// TIA Portal V20 export
FUNCTION_BLOCK "CallEquipment"   // FB36, LAD
TITLE = CallEquipment
AUTHOR : ERsystem_FA2_DH. Kim
// This block contains the logic and futher calls (e.g. sequences, control modules, diagnostics etc.) of the equipment module.
// stored: IsIECCheckEnabled true, MemoryReserve 100, Namespace Unit1.Em3, SetENOAutomatically false
   VAR_INPUT
      ZoneOperationEnable { ExternalWritable := 'False'} : "LWONIK_typeSafetyZoneManualOperation";
   END_VAR
   VAR_IN_OUT
      unitStatus : "LAF_typeUnitStatus";   // Current unit status o be used in this EM
      unitAlarmDB : "LAF_typeAlarms";   // Summarized EM Alarms for the Unit
      emFeedback : "LUC_typeEmFeedback";   // Feedback of the EM to the Unit
   END_VAR
   VAR
      InstSequenceWebGuide : "Unit1.Em3.Sequence_1_WebGuide";
      instWebGuideHomeJob1 { S7_SetPoint := 'True'} : "LAF_SelectJob";
      instWebGuideGuidingJob2 { S7_SetPoint := 'True'} : "LAF_SelectJob";
      instCmSafetyPinIdlePositionSensor : "LBC_DigitalSignalCn";
      instCmIonizerTopMaintDetection { S7_SetPoint := 'True'} : "LBC_DigitalSignalCn";
      instCmIonizerTopErrorDetection { S7_SetPoint := 'True'} : "LBC_DigitalSignalCn";
      instCmIonizerBtmMaintDetection { S7_SetPoint := 'True'} : "LBC_DigitalSignalCn";
      instCmIonizerBtmErrorDetection { S7_SetPoint := 'True'} : "LBC_DigitalSignalCn";
      instCmDancerEncoder { ExternalAccessible := 'False'; ExternalVisible := 'False'; ExternalWritable := 'False'; S7_SetPoint := 'True'} : "LBC_AnalogInputCn";
      instCmLoadCellControllerInterface { ExternalAccessible := 'False'; ExternalVisible := 'False'; ExternalWritable := 'False'; S7_SetPoint := 'True'} : "LBC_AnalogInputCn";
      instCmDancerElectroPneumaticRegulator { ExternalAccessible := 'False'; ExternalVisible := 'False'; ExternalWritable := 'False'; S7_SetPoint := 'True'} : "LBC_AnalogOutputCn";
      instCmCompensatorAxisX { S7_SetPoint := 'True'} : "LBC_Axis64Pos_TecPlcCn";
      instCmUnwinderVirtualAxisX { S7_SetPoint := 'True'} : "LBC_Axis64Pos_TecPlcCn";
      instInterlockCompensatorAxisX { S7_SetPoint := 'True'} : "LER_Axis64Pos_InterlockSummary";
      instInterlockUnwinderVirtualAxisX { S7_SetPoint := 'True'} : "LER_Axis64Pos_InterlockSummary";
      instCmDancerFwdBwd { ExternalAccessible := 'False'; ExternalVisible := 'False'; ExternalWritable := 'False'; S7_SetPoint := 'True'} : "LBC_TwoWayActuatorCn";
      instCmSepaUnwinderIonizerTop { ExternalAccessible := 'False'; ExternalVisible := 'False'; ExternalWritable := 'False'; S7_SetPoint := 'True'} : "LBC_TwoWayActuatorCn";
      instCmSepaUnwinderIonizerBottom { ExternalAccessible := 'False'; ExternalVisible := 'False'; ExternalWritable := 'False'; S7_SetPoint := 'True'} : "LBC_TwoWayActuatorCn";
      instCmEpcPivot { ExternalAccessible := 'False'; ExternalVisible := 'False'; ExternalWritable := 'False'; S7_SetPoint := 'True'} : "LER_EPC_CON600";
      instManageAlarms { ExternalWritable := 'False'} : "LAF_ManageAlarms";
      instEventsPFE : "Unit1.Em3.EventsPFE";
      statUnitStatus { ExternalWritable := 'False'} : "LAF_typeUnitStatus";   // Unit Status used in this EM
      statSlmStatus : Struct
         running { ExternalWritable := 'False'} : Bool;
         powerOff { ExternalWritable := 'False'} : Bool;
      END_STRUCT;
      statTonTime { ExternalAccessible := 'False'; ExternalVisible := 'False'; ExternalWritable := 'False'} : Array[0..1999] of TON_TIME;
      statTofTime { ExternalAccessible := 'False'; ExternalVisible := 'False'; ExternalWritable := 'False'} : Array[0..99] of TOF_TIME;
      statPulse { ExternalAccessible := 'False'; ExternalVisible := 'False'; ExternalWritable := 'False'} : Struct
         miscellaneous : Array[0..99] of Bool;
         workingDone : Struct
            mainPnP : Array[0..99] of Bool;
            alignTable : Array[0..99] of Bool;
            ngPnP : Array[0..99] of Bool;
         END_STRUCT;
         axisEnable : Array[0..99] of Bool;
         brakeTest : Array[0..99] of Bool;
      END_STRUCT;
      statEnableManualCmds : Bool;
      Scan_on : Bool;
      "*** Interlock Axis ***" { ExternalAccessible := 'False'; ExternalVisible := 'False'; ExternalWritable := 'False'} : Bool;
      "compenastor X Home" { S7_SetPoint := 'True'} : "Homing.LER_Axis";
      "compenastor X Jog_CW" { S7_SetPoint := 'True'} : "Jog.LER_Axis";
      "compenastor X Jog_CCW" { S7_SetPoint := 'True'} : "Jog.LER_Axis";
      "compenastor X Position_" { S7_SetPoint := 'True'} : Array[0..5] of "Position.LER_Axis";
      "*** Interlock Actuator ******" { ExternalAccessible := 'False'; ExternalVisible := 'False'; ExternalWritable := 'False'} : Bool;
      "DancerFwdBwd Home" { S7_SetPoint := 'True'} : "Cylinder.LER_Actuator";
      "DancerFwdBwd Work" { S7_SetPoint := 'True'} : "Cylinder.LER_Actuator";
      "SepaUnwinderIonizer Home" { S7_SetPoint := 'True'} : "Cylinder.LER_Actuator";
      "SepaUnwinderIonizer Work" { S7_SetPoint := 'True'} : "Cylinder.LER_Actuator";
      "SepaUnwinderIonizerBottom Home" { S7_SetPoint := 'True'} : "Cylinder.LER_Actuator";
      "SepaUnwinderIonizerBottom Work" { S7_SetPoint := 'True'} : "Cylinder.LER_Actuator";
      AXIS3 : "LER_CM_Name";
      Cylinder10 : "LER_CM_Name";
      instCmRotaionSafetyPinPositionSensor { ExternalAccessible := 'False'; ExternalVisible := 'False'; ExternalWritable := 'False'} : "LBC_DigitalSignalCn";
      citi_Ptrig : Array[0..20] of Bool;
      citiTon : Array[0..20] of TON_TIME;
      citi : Time;
      citiTest : Array[0..20] of Bool;
   END_VAR
   VAR_TEMP
      tempIndex : Int;
      tempScInProduction : Bool;   // Mode Production and StateComplete
      tempScNoProduction : Bool;   // Mode Manual and StateComplete
   END_VAR
   VAR CONSTANT
      delayTime : Time := T#3s;
      TRUE : Bool := TRUE;
      FALSE : Bool := FALSE;
      NO_JOB : DInt;   // No job
      MIN_POSITION_NUMBER : SInt;
      INIT_POSITION_NUMBER : SInt := -1;
   END_VAR
   // // instCmCompensatorAxisX.instAxisCtrl.configuration.posAbsolute.positionChangeOnTheFly : TRUE: Changing position on-the-fly; FALSE: Position change requires a new rising edge at source.posAbsolute input
   // // instCmCompensatorAxisX.instAxisCtrl.configuration.posAbsolute.velocityChangeOnTheFly : TRUE: Changing velocity on-the-fly; FALSE: Velocity change requires a new rising edge at source.posAbsolute input
   // // instCmCompensatorAxisX.statCurrentInputs.posAbsolute : Internal storage for edge detection of source.posAbsolute
   // // instCmCompensatorAxisX.statPreviousInputs.posAbsolute : Internal storage for edge detection of source.posAbsolute
   // // instCmCompensatorAxisX.statCurrentInterface.posAbsolute : Internal storage for edge detection of source.posAbsolute
   // // instCmCompensatorAxisX.statPreviousInterface.posAbsolute : Internal storage for edge detection of source.posAbsolute
   // // instCmUnwinderVirtualAxisX.instAxisCtrl.configuration.posAbsolute.positionChangeOnTheFly : TRUE: Changing position on-the-fly; FALSE: Position change requires a new rising edge at source.posAbsolute input
   // // instCmUnwinderVirtualAxisX.instAxisCtrl.configuration.posAbsolute.velocityChangeOnTheFly : TRUE: Changing velocity on-the-fly; FALSE: Velocity change requires a new rising edge at source.posAbsolute input
   // // instCmUnwinderVirtualAxisX.statCurrentInputs.posAbsolute : Internal storage for edge detection of source.posAbsolute
   // // instCmUnwinderVirtualAxisX.statPreviousInputs.posAbsolute : Internal storage for edge detection of source.posAbsolute
   // // instCmUnwinderVirtualAxisX.statCurrentInterface.posAbsolute : Internal storage for edge detection of source.posAbsolute
   // // instCmUnwinderVirtualAxisX.statPreviousInterface.posAbsolute : Internal storage for edge detection of source.posAbsolute
   VAR_TEMP   // added for the SCL form of the ladder/FBD networks
      _w1 : Bool;
      _w2 : Bool;
      _w3 : Bool;
      _w4 : Bool;
      _w5 : Bool;
      _w6 : Bool;
      _w7 : Bool;
      _w8 : Bool;
      _w9 : Bool;
   END_VAR
BEGIN

REGION Network 1: BLOCK INFO HEADER
   // (company) / (C) Copyright (year)
   // ---------------------------------------------------------------------------------
   // Title:                             (Title of this block)
   // Comment/Function: (that is implemented in the block)
   // Library/Family:           (that the source is dedicated to)
   // Author:                        (department / person in charge / contact)
   // Target System:          (test system with FW version)
   // Engineering:              TIA Portal (SW version)
   // Restrictions:               (OB types, etc.)
   // Requirements:           (hardware, technological package, etc.)
   // ---------------------------------------------------------------------------------
   // Change log table:
   // Version          | Date             | Signature      | Expert in charge  | Changes applied ------------------------|----------------------|-------------------------|--------------------------------|-----------------------
   // 001.000.000 | yyyy-mm-dd | 0x00000000 | (name of expert) | First released version
END_REGION

REGION Network 2: DESCRIPTION
   // This is a template block provided by the Automation Framework. It can be used to create an own project.
   // The Block Info Header is prepared to put in your own data.
   // Description of the block could be added here and the docu created by Code2Docu.
END_REGION

REGION Network 3: TRUE: Disable the monitoring of the Home position feedback. FALSE: Home position is reached after `monitoringReachingFeedback` time expires.
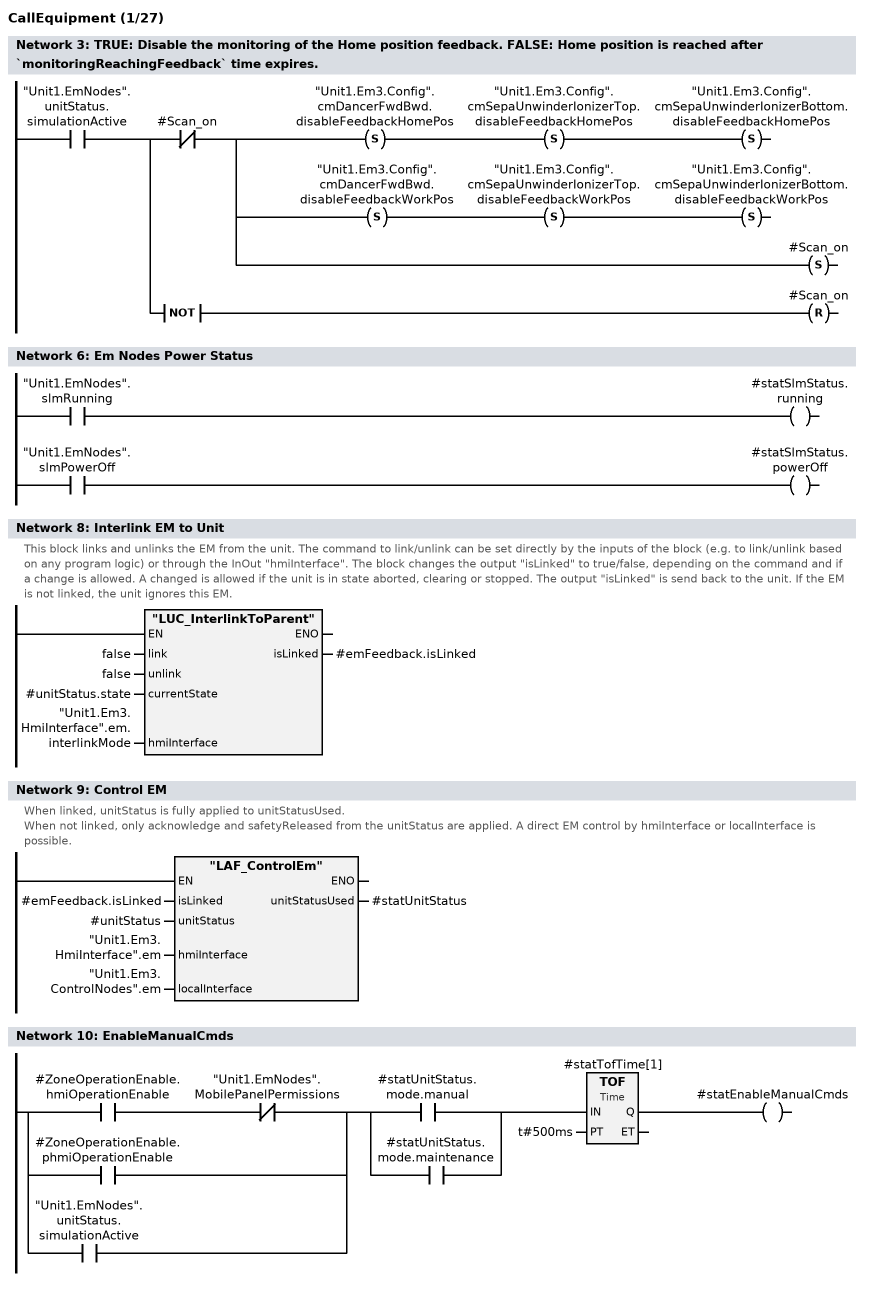
   RUNG wire#powerrail
      Contact( "Unit1.EmNodes".unitStatus.simulationActive )
      wire#w1
      I_Contact( #Scan_on )
      wire#w2
      S_Coil( "Unit1.Em3.Config".cmDancerFwdBwd.disableFeedbackHomePos )
      S_Coil( "Unit1.Em3.Config".cmSepaUnwinderIonizerTop.disableFeedbackHomePos )
      S_Coil( "Unit1.Em3.Config".cmSepaUnwinderIonizerBottom.disableFeedbackHomePos )
   END_RUNG
   RUNG wire#w2
      S_Coil( "Unit1.Em3.Config".cmDancerFwdBwd.disableFeedbackWorkPos )
      S_Coil( "Unit1.Em3.Config".cmSepaUnwinderIonizerTop.disableFeedbackWorkPos )
      S_Coil( "Unit1.Em3.Config".cmSepaUnwinderIonizerBottom.disableFeedbackWorkPos )
   END_RUNG
   RUNG wire#w2
      S_Coil( #Scan_on )
   END_RUNG
   RUNG wire#w1
      Not()
      R_Coil( #Scan_on )
   END_RUNG
   // the same network as SCL:
   IF "Unit1.EmNodes".unitStatus.simulationActive AND NOT #Scan_on THEN
       "Unit1.Em3.Config".cmDancerFwdBwd.disableFeedbackHomePos := TRUE;
       "Unit1.Em3.Config".cmSepaUnwinderIonizerTop.disableFeedbackHomePos := TRUE;
       "Unit1.Em3.Config".cmSepaUnwinderIonizerBottom.disableFeedbackHomePos := TRUE;
       "Unit1.Em3.Config".cmDancerFwdBwd.disableFeedbackWorkPos := TRUE;
       "Unit1.Em3.Config".cmSepaUnwinderIonizerTop.disableFeedbackWorkPos := TRUE;
       "Unit1.Em3.Config".cmSepaUnwinderIonizerBottom.disableFeedbackWorkPos := TRUE;
       #Scan_on := TRUE;
   END_IF;
   IF NOT "Unit1.EmNodes".unitStatus.simulationActive THEN #Scan_on := FALSE; END_IF;
END_REGION

REGION Network 4: ******************** Unit Input ********************
END_REGION

REGION Network 5: Em2 Sequence Interface
END_REGION

REGION Network 6: Em Nodes Power Status
   RUNG wire#powerrail
      Contact( "Unit1.EmNodes".slmRunning )
      Coil( #statSlmStatus.running )
   END_RUNG
   RUNG wire#powerrail
      Contact( "Unit1.EmNodes".slmPowerOff )
      Coil( #statSlmStatus.powerOff )
   END_RUNG
   // the same network as SCL:
   #statSlmStatus.running := "Unit1.EmNodes".slmRunning;
   #statSlmStatus.powerOff := "Unit1.EmNodes".slmPowerOff;
END_REGION

REGION Network 7: *************** Equipment Control **************************
END_REGION

REGION Network 8: Interlink EM to Unit
   // This block links and unlinks the EM from the unit. The command to link/unlink can be set directly by the inputs of the block (e.g. to link/unlink based on any program logic) or through the InOut "hmiInterface". The block changes the output "isLinked" to true/false, depending on the command and if a change is allowed. A changed is allowed if the unit is in state aborted, clearing or stopped. The output "isLinked" is send back to the unit. If the EM is not linked, the unit ignores this EM.
   RUNG wire#powerrail
      "LUC_InterlinkToParent"(link := false, unlink := false, currentState := #unitStatus.state, hmiInterface := "Unit1.Em3.HmiInterface".em.interlinkMode, isLinked => #emFeedback.isLinked)
   END_RUNG
   // the same network as SCL:
   "LUC_InterlinkToParent"(link := false,
                           unlink := false,
                           currentState := #unitStatus.state,
                           hmiInterface := "Unit1.Em3.HmiInterface".em.interlinkMode,
                           isLinked => #emFeedback.isLinked);
END_REGION

REGION Network 9: Control EM
   // When linked, unitStatus is fully applied to unitStatusUsed.
   // When not linked, only acknowledge and safetyReleased from the unitStatus are applied. A direct EM control by hmiInterface or localInterface is possible.
   RUNG wire#powerrail
      "LAF_ControlEm"(isLinked := #emFeedback.isLinked, unitStatus := #unitStatus, hmiInterface := "Unit1.Em3.HmiInterface".em, localInterface := "Unit1.Em3.ControlNodes".em, unitStatusUsed => #statUnitStatus)
   END_RUNG
   // the same network as SCL:
   "LAF_ControlEm"(isLinked := #emFeedback.isLinked,
                   unitStatus := #unitStatus,
                   hmiInterface := "Unit1.Em3.HmiInterface".em,
                   localInterface := "Unit1.Em3.ControlNodes".em,
                   unitStatusUsed => #statUnitStatus);
END_REGION

REGION Network 10: EnableManualCmds
   RUNG wire#powerrail
      Contact( #ZoneOperationEnable.hmiOperationEnable )
      I_Contact( "Unit1.EmNodes".MobilePanelPermissions )
      wire#w1
      Contact( #statUnitStatus.mode.manual )
      wire#w2
      { S7_Templates := "time_type := Time" } #statTofTime[1].TOF(pt := t#500ms, et =>)
      Coil( #statEnableManualCmds )
   END_RUNG
   RUNG wire#powerrail
      Contact( #ZoneOperationEnable.phmiOperationEnable )
   END_RUNG wire#w1
   RUNG wire#powerrail
      Contact( "Unit1.EmNodes".unitStatus.simulationActive )
   END_RUNG wire#w1
   RUNG wire#w1
      Contact( #statUnitStatus.mode.maintenance )
   END_RUNG wire#w2
   // the same network as SCL:
   #statTofTime[1].TOF(IN := ((#ZoneOperationEnable.hmiOperationEnable AND NOT "Unit1.EmNodes".MobilePanelPermissions) OR #ZoneOperationEnable.phmiOperationEnable OR "Unit1.EmNodes".unitStatus.simulationActive) AND (#statUnitStatus.mode.manual OR #statUnitStatus.mode.maintenance),
                       PT := t#500ms);
   #statEnableManualCmds := #statTofTime[1].Q;
END_REGION

REGION Network 11: *************** Control Modules (Sensors) ********************
   // Call control modules that are sensors before the em logic (jobs and sequence), so that the latest value is used in the logic.
END_REGION

REGION Network 12: Call cmDancer Safety Pin Idle Position Sensor (LBC_DigitalSignal)
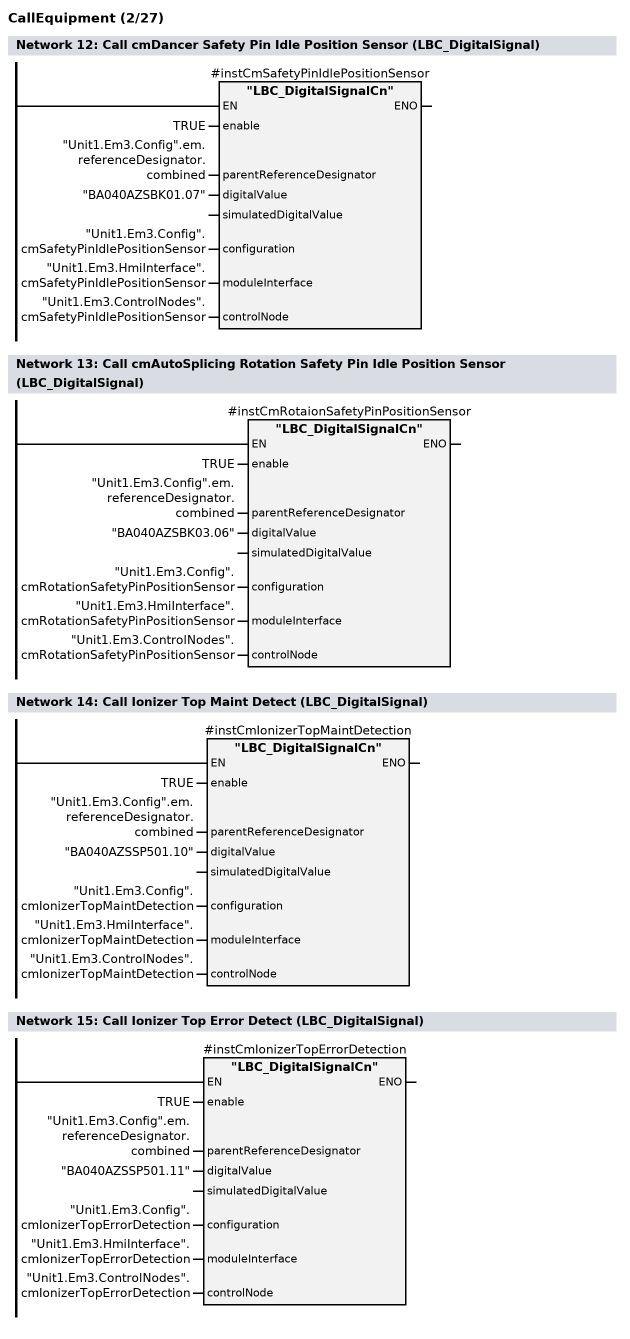
   RUNG wire#powerrail
      #instCmSafetyPinIdlePositionSensor(enable := TRUE, parentReferenceDesignator := "Unit1.Em3.Config".em.referenceDesignator.combined, digitalValue := "BA040AZSBK01.07", simulatedDigitalValue :=, configuration := "Unit1.Em3.Config".cmSafetyPinIdlePositionSensor, moduleInterface := "Unit1.Em3.HmiInterface".cmSafetyPinIdlePositionSensor, controlNode := "Unit1.Em3.ControlNodes".cmSafetyPinIdlePositionSensor)
   END_RUNG
   // the same network as SCL:
   #instCmSafetyPinIdlePositionSensor(enable := TRUE,   // "LBC_DigitalSignalCn"
                           parentReferenceDesignator := "Unit1.Em3.Config".em.referenceDesignator.combined,
                           digitalValue := "BA040AZSBK01.07",
                           configuration := "Unit1.Em3.Config".cmSafetyPinIdlePositionSensor,
                           moduleInterface := "Unit1.Em3.HmiInterface".cmSafetyPinIdlePositionSensor,
                           controlNode := "Unit1.Em3.ControlNodes".cmSafetyPinIdlePositionSensor);
END_REGION

REGION Network 13: Call cmAutoSplicing Rotation Safety Pin Idle Position Sensor (LBC_DigitalSignal)
   RUNG wire#powerrail
      #instCmRotaionSafetyPinPositionSensor(enable := TRUE, parentReferenceDesignator := "Unit1.Em3.Config".em.referenceDesignator.combined, digitalValue := "BA040AZSBK03.06", simulatedDigitalValue :=, configuration := "Unit1.Em3.Config".cmRotationSafetyPinPositionSensor, moduleInterface := "Unit1.Em3.HmiInterface".cmRotationSafetyPinPositionSensor, controlNode := "Unit1.Em3.ControlNodes".cmRotationSafetyPinPositionSensor)
   END_RUNG
   // the same network as SCL:
   #instCmRotaionSafetyPinPositionSensor(enable := TRUE,   // "LBC_DigitalSignalCn"
                           parentReferenceDesignator := "Unit1.Em3.Config".em.referenceDesignator.combined,
                           digitalValue := "BA040AZSBK03.06",
                           configuration := "Unit1.Em3.Config".cmRotationSafetyPinPositionSensor,
                           moduleInterface := "Unit1.Em3.HmiInterface".cmRotationSafetyPinPositionSensor,
                           controlNode := "Unit1.Em3.ControlNodes".cmRotationSafetyPinPositionSensor);
END_REGION

REGION Network 14: Call Ionizer Top Maint Detect (LBC_DigitalSignal)
   RUNG wire#powerrail
      #instCmIonizerTopMaintDetection(enable := TRUE, parentReferenceDesignator := "Unit1.Em3.Config".em.referenceDesignator.combined, digitalValue := "BA040AZSSP501.10", simulatedDigitalValue :=, configuration := "Unit1.Em3.Config".cmIonizerTopMaintDetection, moduleInterface := "Unit1.Em3.HmiInterface".cmIonizerTopMaintDetection, controlNode := "Unit1.Em3.ControlNodes".cmIonizerTopMaintDetection)
   END_RUNG
   // the same network as SCL:
   #instCmIonizerTopMaintDetection(enable := TRUE,   // "LBC_DigitalSignalCn"
                           parentReferenceDesignator := "Unit1.Em3.Config".em.referenceDesignator.combined,
                           digitalValue := "BA040AZSSP501.10",
                           configuration := "Unit1.Em3.Config".cmIonizerTopMaintDetection,
                           moduleInterface := "Unit1.Em3.HmiInterface".cmIonizerTopMaintDetection,
                           controlNode := "Unit1.Em3.ControlNodes".cmIonizerTopMaintDetection);
END_REGION

REGION Network 15: Call Ionizer Top Error Detect (LBC_DigitalSignal)
   RUNG wire#powerrail
      #instCmIonizerTopErrorDetection(enable := TRUE, parentReferenceDesignator := "Unit1.Em3.Config".em.referenceDesignator.combined, digitalValue := "BA040AZSSP501.11", simulatedDigitalValue :=, configuration := "Unit1.Em3.Config".cmIonizerTopErrorDetection, moduleInterface := "Unit1.Em3.HmiInterface".cmIonizerTopErrorDetection, controlNode := "Unit1.Em3.ControlNodes".cmIonizerTopErrorDetection)
   END_RUNG
   // the same network as SCL:
   #instCmIonizerTopErrorDetection(enable := TRUE,   // "LBC_DigitalSignalCn"
                           parentReferenceDesignator := "Unit1.Em3.Config".em.referenceDesignator.combined,
                           digitalValue := "BA040AZSSP501.11",
                           configuration := "Unit1.Em3.Config".cmIonizerTopErrorDetection,
                           moduleInterface := "Unit1.Em3.HmiInterface".cmIonizerTopErrorDetection,
                           controlNode := "Unit1.Em3.ControlNodes".cmIonizerTopErrorDetection);
END_REGION

REGION Network 16: Call Ionizer Btm Maint Detect (LBC_DigitalSignal)
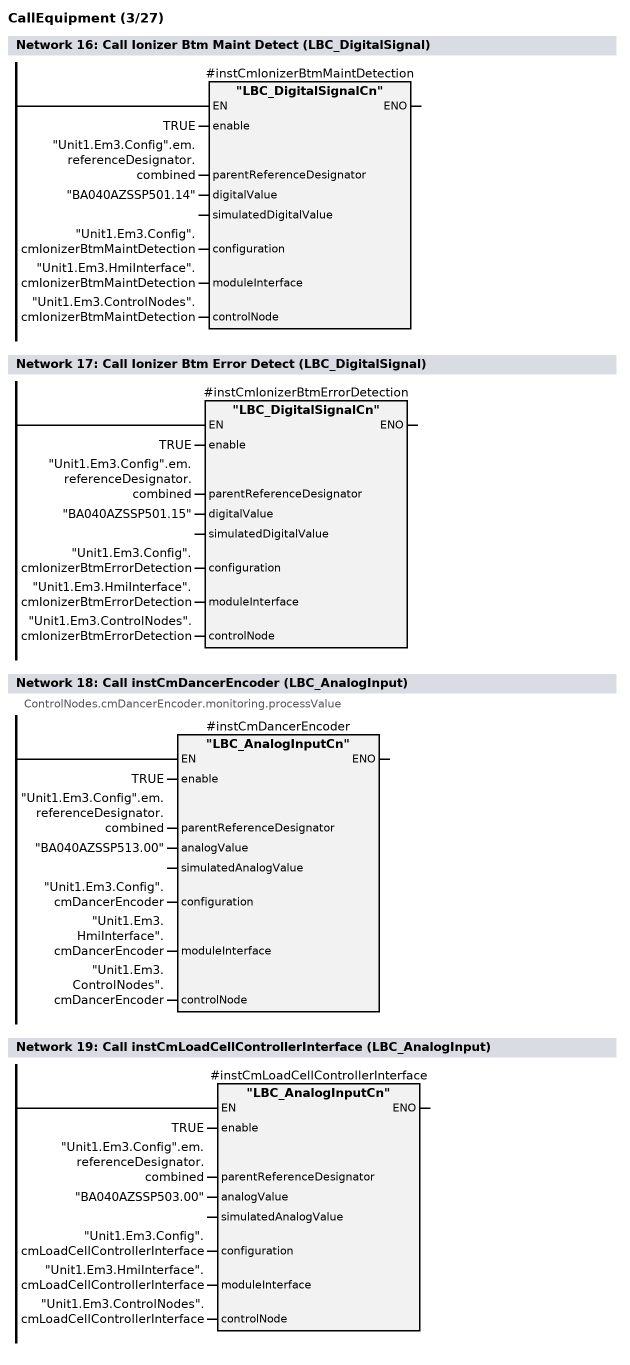
   RUNG wire#powerrail
      #instCmIonizerBtmMaintDetection(enable := TRUE, parentReferenceDesignator := "Unit1.Em3.Config".em.referenceDesignator.combined, digitalValue := "BA040AZSSP501.14", simulatedDigitalValue :=, configuration := "Unit1.Em3.Config".cmIonizerBtmMaintDetection, moduleInterface := "Unit1.Em3.HmiInterface".cmIonizerBtmMaintDetection, controlNode := "Unit1.Em3.ControlNodes".cmIonizerBtmMaintDetection)
   END_RUNG
   // the same network as SCL:
   #instCmIonizerBtmMaintDetection(enable := TRUE,   // "LBC_DigitalSignalCn"
                           parentReferenceDesignator := "Unit1.Em3.Config".em.referenceDesignator.combined,
                           digitalValue := "BA040AZSSP501.14",
                           configuration := "Unit1.Em3.Config".cmIonizerBtmMaintDetection,
                           moduleInterface := "Unit1.Em3.HmiInterface".cmIonizerBtmMaintDetection,
                           controlNode := "Unit1.Em3.ControlNodes".cmIonizerBtmMaintDetection);
END_REGION

REGION Network 17: Call Ionizer Btm Error Detect (LBC_DigitalSignal)
   RUNG wire#powerrail
      #instCmIonizerBtmErrorDetection(enable := TRUE, parentReferenceDesignator := "Unit1.Em3.Config".em.referenceDesignator.combined, digitalValue := "BA040AZSSP501.15", simulatedDigitalValue :=, configuration := "Unit1.Em3.Config".cmIonizerBtmErrorDetection, moduleInterface := "Unit1.Em3.HmiInterface".cmIonizerBtmErrorDetection, controlNode := "Unit1.Em3.ControlNodes".cmIonizerBtmErrorDetection)
   END_RUNG
   // the same network as SCL:
   #instCmIonizerBtmErrorDetection(enable := TRUE,   // "LBC_DigitalSignalCn"
                           parentReferenceDesignator := "Unit1.Em3.Config".em.referenceDesignator.combined,
                           digitalValue := "BA040AZSSP501.15",
                           configuration := "Unit1.Em3.Config".cmIonizerBtmErrorDetection,
                           moduleInterface := "Unit1.Em3.HmiInterface".cmIonizerBtmErrorDetection,
                           controlNode := "Unit1.Em3.ControlNodes".cmIonizerBtmErrorDetection);
END_REGION

REGION Network 18: Call instCmDancerEncoder (LBC_AnalogInput)
   // ControlNodes.cmDancerEncoder.monitoring.processValue
   RUNG wire#powerrail
      #instCmDancerEncoder(enable := TRUE, parentReferenceDesignator := "Unit1.Em3.Config".em.referenceDesignator.combined, analogValue := "BA040AZSSP513.00", simulatedAnalogValue :=, configuration := "Unit1.Em3.Config".cmDancerEncoder, moduleInterface := "Unit1.Em3.HmiInterface".cmDancerEncoder, controlNode := "Unit1.Em3.ControlNodes".cmDancerEncoder)
   END_RUNG
   // the same network as SCL:
   #instCmDancerEncoder(enable := TRUE,   // "LBC_AnalogInputCn"
                        parentReferenceDesignator := "Unit1.Em3.Config".em.referenceDesignator.combined,
                        analogValue := "BA040AZSSP513.00",
                        configuration := "Unit1.Em3.Config".cmDancerEncoder,
                        moduleInterface := "Unit1.Em3.HmiInterface".cmDancerEncoder,
                        controlNode := "Unit1.Em3.ControlNodes".cmDancerEncoder);
END_REGION

REGION Network 19: Call instCmLoadCellControllerInterface (LBC_AnalogInput)
   RUNG wire#powerrail
      #instCmLoadCellControllerInterface(enable := TRUE, parentReferenceDesignator := "Unit1.Em3.Config".em.referenceDesignator.combined, analogValue := "BA040AZSSP503.00", simulatedAnalogValue :=, configuration := "Unit1.Em3.Config".cmLoadCellControllerInterface, moduleInterface := "Unit1.Em3.HmiInterface".cmLoadCellControllerInterface, controlNode := "Unit1.Em3.ControlNodes".cmLoadCellControllerInterface)
   END_RUNG
   // the same network as SCL:
   #instCmLoadCellControllerInterface(enable := TRUE,   // "LBC_AnalogInputCn"
                           parentReferenceDesignator := "Unit1.Em3.Config".em.referenceDesignator.combined,
                           analogValue := "BA040AZSSP503.00",
                           configuration := "Unit1.Em3.Config".cmLoadCellControllerInterface,
                           moduleInterface := "Unit1.Em3.HmiInterface".cmLoadCellControllerInterface,
                           controlNode := "Unit1.Em3.ControlNodes".cmLoadCellControllerInterface);
END_REGION

REGION Network 20: Call instCmDancerElectroPneumaticRegulator (LBC_AnalogOutput)
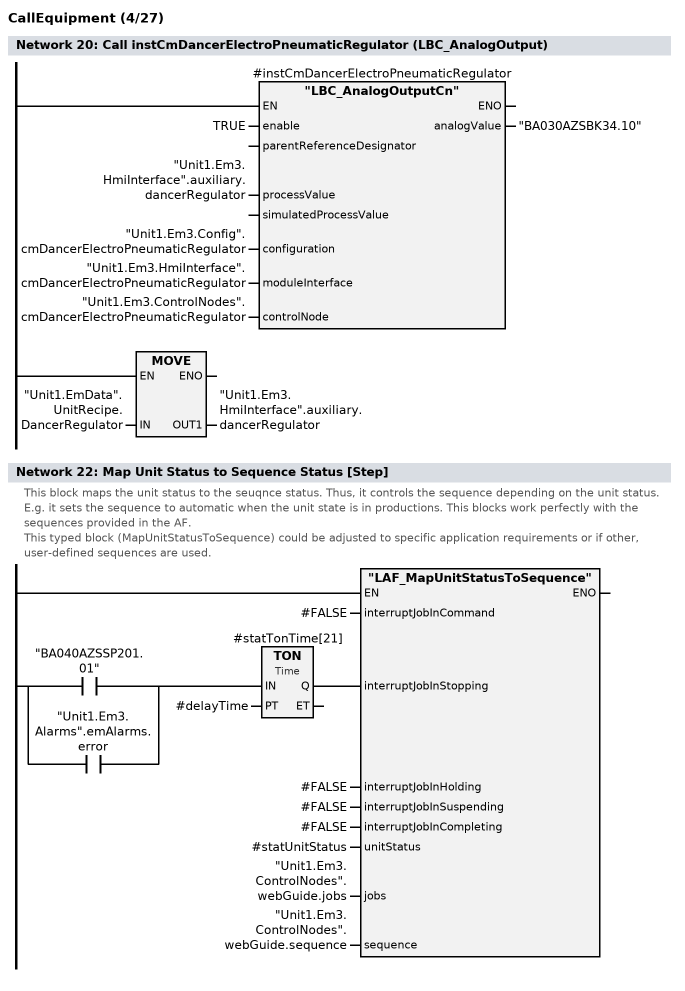
   RUNG wire#powerrail
      #instCmDancerElectroPneumaticRegulator(enable := TRUE, parentReferenceDesignator :=, processValue := "Unit1.Em3.HmiInterface".auxiliary.dancerRegulator, simulatedProcessValue :=, configuration := "Unit1.Em3.Config".cmDancerElectroPneumaticRegulator, moduleInterface := "Unit1.Em3.HmiInterface".cmDancerElectroPneumaticRegulator, controlNode := "Unit1.Em3.ControlNodes".cmDancerElectroPneumaticRegulator, analogValue => "BA030AZSBK34.10")
   END_RUNG
   RUNG wire#powerrail
      Move(in := "Unit1.EmData".UnitRecipe.DancerRegulator, out1 => "Unit1.Em3.HmiInterface".auxiliary.dancerRegulator)
   END_RUNG
   // the same network as SCL:
   #instCmDancerElectroPneumaticRegulator(enable := TRUE,   // "LBC_AnalogOutputCn"
                           processValue := "Unit1.Em3.HmiInterface".auxiliary.dancerRegulator,
                           configuration := "Unit1.Em3.Config".cmDancerElectroPneumaticRegulator,
                           moduleInterface := "Unit1.Em3.HmiInterface".cmDancerElectroPneumaticRegulator,
                           controlNode := "Unit1.Em3.ControlNodes".cmDancerElectroPneumaticRegulator,
                           analogValue => "BA030AZSBK34.10");
   "Unit1.Em3.HmiInterface".auxiliary.dancerRegulator := "Unit1.EmData".UnitRecipe.DancerRegulator;
END_REGION

REGION Network 21: *************** Equipment Logic ***************************
END_REGION

REGION Network 22: Map Unit Status to Sequence Status [Step]
   // This block maps the unit status to the seuqnce status. Thus, it controls the sequence depending on the unit status. E.g. it sets the sequence to automatic when the unit state is in productions. This blocks work perfectly with the sequences provided in the AF. 
   // This typed block (MapUnitStatusToSequence) could be adjusted to specific application requirements or if other, user-defined sequences are used.
   RUNG wire#powerrail
      "LAF_MapUnitStatusToSequence"(interruptJobInStopping := wire#w2, interruptJobInCommand := #FALSE, interruptJobInHolding := #FALSE, interruptJobInSuspending := #FALSE, interruptJobInCompleting := #FALSE, unitStatus := #statUnitStatus, jobs := "Unit1.Em3.ControlNodes".webGuide.jobs, sequence := "Unit1.Em3.ControlNodes".webGuide.sequence)
   END_RUNG
   RUNG wire#powerrail
      Contact( "BA040AZSSP201.01" )
      wire#w1
      { S7_Templates := "time_type := Time" } #statTonTime[21].TON(pt := #delayTime, et =>)
   END_RUNG wire#w2
   RUNG wire#powerrail
      Contact( "Unit1.Em3.Alarms".emAlarms.error )
   END_RUNG wire#w1
   // the same network as SCL:
   #statTonTime[21].TON(IN := "BA040AZSSP201.01" OR "Unit1.Em3.Alarms".emAlarms.error, PT := #delayTime);
   "LAF_MapUnitStatusToSequence"(interruptJobInCommand := #FALSE,
                           interruptJobInStopping := #statTonTime[21].Q,
                           interruptJobInHolding := #FALSE,
                           interruptJobInSuspending := #FALSE,
                           interruptJobInCompleting := #FALSE,
                           unitStatus := #statUnitStatus,
                           jobs := "Unit1.Em3.ControlNodes".webGuide.jobs,
                           sequence := "Unit1.Em3.ControlNodes".webGuide.sequence);
END_REGION

REGION Network 24: Web Guide Select Job
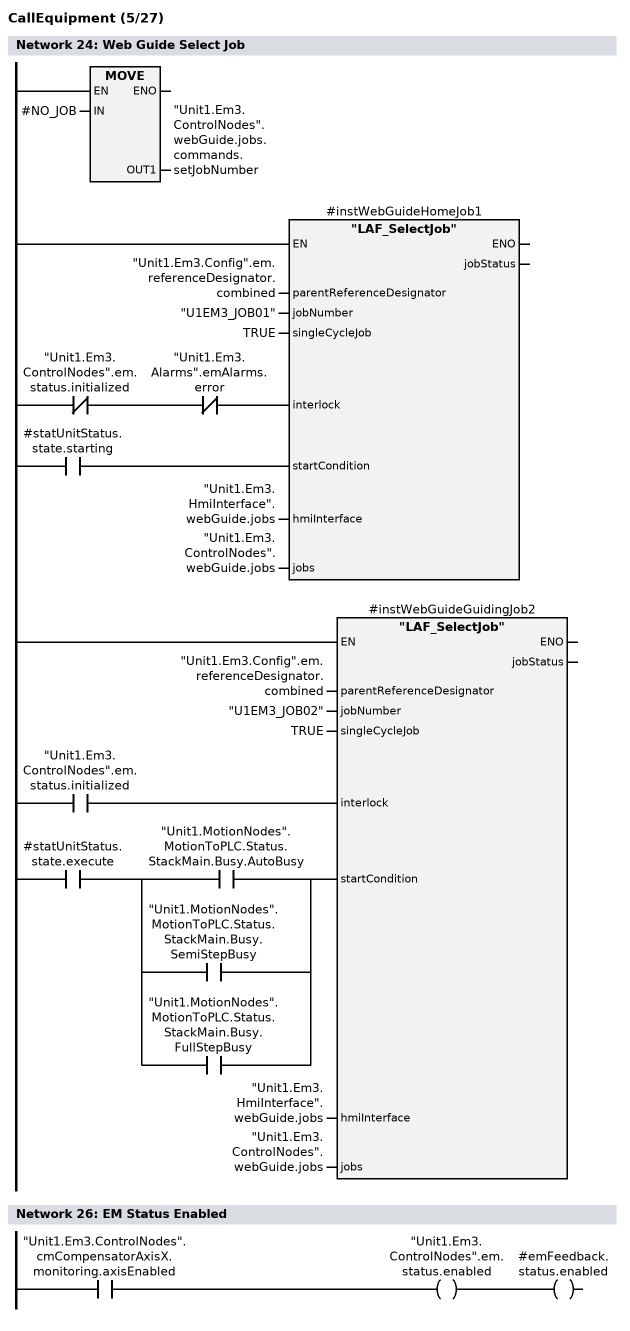
   RUNG wire#powerrail
      Move(in := #NO_JOB, out1 => "Unit1.Em3.ControlNodes".webGuide.jobs.commands.setJobNumber)
   END_RUNG
   RUNG wire#powerrail
      #instWebGuideHomeJob1(interlock := wire#w1, startCondition := wire#w2, parentReferenceDesignator := "Unit1.Em3.Config".em.referenceDesignator.combined, jobNumber := "U1EM3_JOB01", singleCycleJob := TRUE, hmiInterface := "Unit1.Em3.HmiInterface".webGuide.jobs, jobs := "Unit1.Em3.ControlNodes".webGuide.jobs, jobStatus =>)
   END_RUNG
   RUNG wire#powerrail
      I_Contact( "Unit1.Em3.ControlNodes".em.status.initialized )
      I_Contact( "Unit1.Em3.Alarms".emAlarms.error )
   END_RUNG wire#w1
   RUNG wire#powerrail
      Contact( #statUnitStatus.state.starting )
   END_RUNG wire#w2
   RUNG wire#powerrail
      #instWebGuideGuidingJob2(interlock := wire#w3, startCondition := wire#w5, parentReferenceDesignator := "Unit1.Em3.Config".em.referenceDesignator.combined, jobNumber := "U1EM3_JOB02", singleCycleJob := TRUE, hmiInterface := "Unit1.Em3.HmiInterface".webGuide.jobs, jobs := "Unit1.Em3.ControlNodes".webGuide.jobs, jobStatus =>)
   END_RUNG
   RUNG wire#powerrail
      Contact( "Unit1.Em3.ControlNodes".em.status.initialized )
   END_RUNG wire#w3
   RUNG wire#powerrail
      Contact( #statUnitStatus.state.execute )
      wire#w4
      Contact( "Unit1.MotionNodes".MotionToPLC.Status.StackMain.Busy.AutoBusy )
   END_RUNG wire#w5
   RUNG wire#w4
      Contact( "Unit1.MotionNodes".MotionToPLC.Status.StackMain.Busy.SemiStepBusy )
   END_RUNG wire#w5
   RUNG wire#w4
      Contact( "Unit1.MotionNodes".MotionToPLC.Status.StackMain.Busy.FullStepBusy )
   END_RUNG wire#w5
   // the same network as SCL:
   "Unit1.Em3.ControlNodes".webGuide.jobs.commands.setJobNumber := #NO_JOB;
   #instWebGuideHomeJob1(parentReferenceDesignator := "Unit1.Em3.Config".em.referenceDesignator.combined,   // "LAF_SelectJob"
                         jobNumber := "U1EM3_JOB01",
                         singleCycleJob := TRUE,
                         interlock := NOT "Unit1.Em3.ControlNodes".em.status.initialized AND NOT "Unit1.Em3.Alarms".emAlarms.error,
                         startCondition := #statUnitStatus.state.starting,
                         hmiInterface := "Unit1.Em3.HmiInterface".webGuide.jobs,
                         jobs := "Unit1.Em3.ControlNodes".webGuide.jobs);
   #instWebGuideGuidingJob2(parentReferenceDesignator := "Unit1.Em3.Config".em.referenceDesignator.combined,   // "LAF_SelectJob"
                           jobNumber := "U1EM3_JOB02",
                           singleCycleJob := TRUE,
                           interlock := "Unit1.Em3.ControlNodes".em.status.initialized,
                           startCondition := #statUnitStatus.state.execute AND ("Unit1.MotionNodes".MotionToPLC.Status.StackMain.Busy.AutoBusy OR "Unit1.MotionNodes".MotionToPLC.Status.StackMain.Busy.SemiStepBusy OR "Unit1.MotionNodes".MotionToPLC.Status.StackMain.Busy.FullStepBusy),
                           hmiInterface := "Unit1.Em3.HmiInterface".webGuide.jobs,
                           jobs := "Unit1.Em3.ControlNodes".webGuide.jobs);
END_REGION

REGION Network 26: EM Status Enabled
   RUNG wire#powerrail
      Contact( "Unit1.Em3.ControlNodes".cmCompensatorAxisX.monitoring.axisEnabled )
      Coil( "Unit1.Em3.ControlNodes".em.status.enabled )
      Coil( #emFeedback.status.enabled )
   END_RUNG
   // the same network as SCL:
   "Unit1.Em3.ControlNodes".em.status.enabled := "Unit1.Em3.ControlNodes".cmCompensatorAxisX.monitoring.axisEnabled;
   #emFeedback.status.enabled := "Unit1.Em3.ControlNodes".cmCompensatorAxisX.monitoring.axisEnabled;
END_REGION

REGION Network 27: Set EM To Initialized
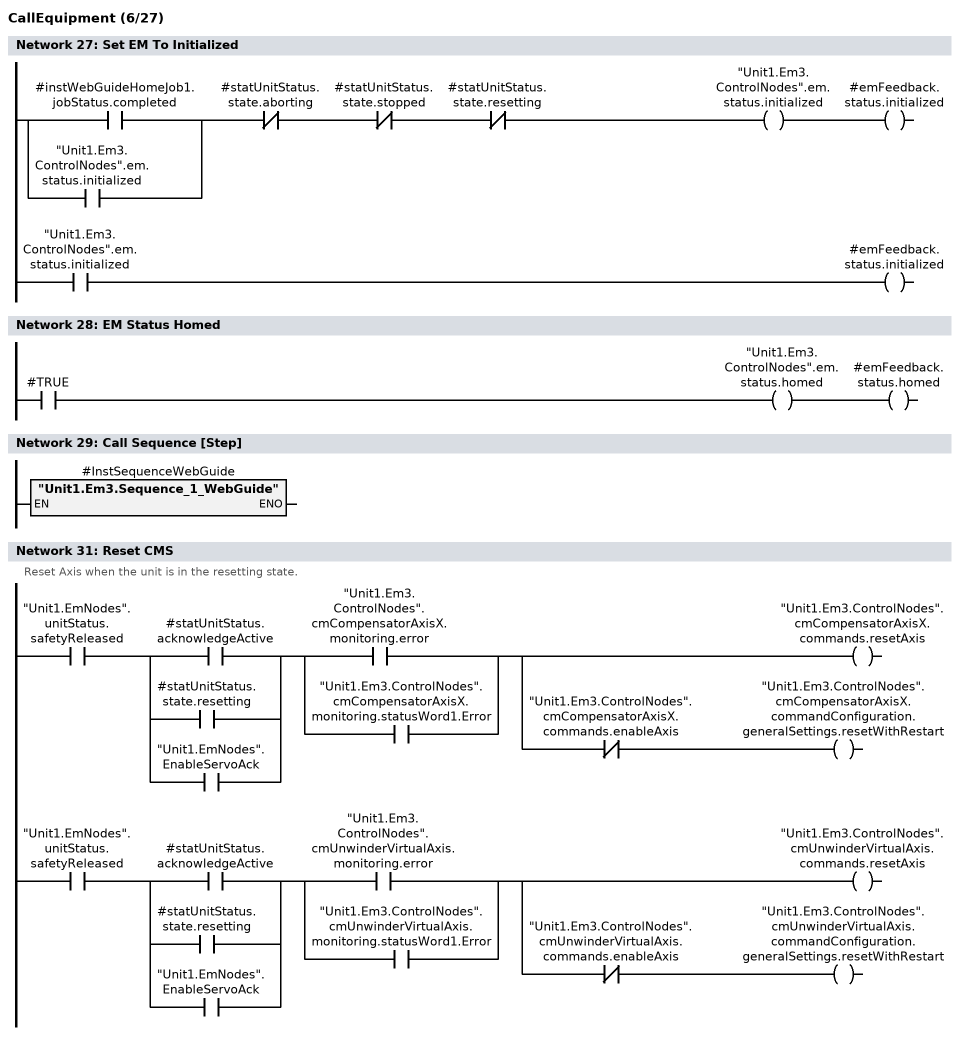
   RUNG wire#powerrail
      Contact( #instWebGuideHomeJob1.jobStatus.completed )
      wire#w1
      I_Contact( #statUnitStatus.state.aborting )
      I_Contact( #statUnitStatus.state.stopped )
      I_Contact( #statUnitStatus.state.resetting )
      Coil( "Unit1.Em3.ControlNodes".em.status.initialized )
      Coil( #emFeedback.status.initialized )
   END_RUNG
   RUNG wire#powerrail
      Contact( "Unit1.Em3.ControlNodes".em.status.initialized )
   END_RUNG wire#w1
   RUNG wire#powerrail
      Contact( "Unit1.Em3.ControlNodes".em.status.initialized )
      Coil( #emFeedback.status.initialized )
   END_RUNG
   // the same network as SCL:
   "Unit1.Em3.ControlNodes".em.status.initialized := (#instWebGuideHomeJob1.jobStatus.completed OR "Unit1.Em3.ControlNodes".em.status.initialized) AND NOT #statUnitStatus.state.aborting AND NOT #statUnitStatus.state.stopped AND NOT #statUnitStatus.state.resetting;
   #emFeedback.status.initialized := "Unit1.Em3.ControlNodes".em.status.initialized;
   #emFeedback.status.initialized := "Unit1.Em3.ControlNodes".em.status.initialized;
END_REGION

REGION Network 28: EM Status Homed
   RUNG wire#powerrail
      Contact( #TRUE )
      Coil( "Unit1.Em3.ControlNodes".em.status.homed )
      Coil( #emFeedback.status.homed )
   END_RUNG
   // the same network as SCL:
   "Unit1.Em3.ControlNodes".em.status.homed := #TRUE;
   #emFeedback.status.homed := #TRUE;
END_REGION

REGION Network 29: Call Sequence [Step]
   RUNG wire#powerrail
      #InstSequenceWebGuide()
   END_RUNG
   // the same network as SCL:
   #InstSequenceWebGuide();   // "Unit1.Em3.Sequence_1_WebGuide"
END_REGION

REGION Network 30: *************** Control Modules (Axis) *******************
   // Call control modules that are actuators after the em logic (jobs and sequence), so that the latest commands are applied to the actuators.
END_REGION

REGION Network 31: Reset CMS
   // Reset Axis when the unit is in the resetting state.
   RUNG wire#powerrail
      Contact( "Unit1.EmNodes".unitStatus.safetyReleased )
      wire#w1
      Contact( #statUnitStatus.acknowledgeActive )
      wire#w2
      Contact( "Unit1.Em3.ControlNodes".cmCompensatorAxisX.monitoring.error )
      wire#w3
      Coil( "Unit1.Em3.ControlNodes".cmCompensatorAxisX.commands.resetAxis )
   END_RUNG
   RUNG wire#w1
      Contact( #statUnitStatus.state.resetting )
   END_RUNG wire#w2
   RUNG wire#w1
      Contact( "Unit1.EmNodes".EnableServoAck )
   END_RUNG wire#w2
   RUNG wire#w2
      Contact( "Unit1.Em3.ControlNodes".cmCompensatorAxisX.monitoring.statusWord1.Error )
   END_RUNG wire#w3
   RUNG wire#w3
      I_Contact( "Unit1.Em3.ControlNodes".cmCompensatorAxisX.commands.enableAxis )
      Coil( "Unit1.Em3.ControlNodes".cmCompensatorAxisX.commandConfiguration.generalSettings.resetWithRestart )
   END_RUNG
   RUNG wire#powerrail
      Contact( "Unit1.EmNodes".unitStatus.safetyReleased )
      wire#w4
      Contact( #statUnitStatus.acknowledgeActive )
      wire#w5
      Contact( "Unit1.Em3.ControlNodes".cmUnwinderVirtualAxis.monitoring.error )
      wire#w6
      Coil( "Unit1.Em3.ControlNodes".cmUnwinderVirtualAxis.commands.resetAxis )
   END_RUNG
   RUNG wire#w4
      Contact( #statUnitStatus.state.resetting )
   END_RUNG wire#w5
   RUNG wire#w4
      Contact( "Unit1.EmNodes".EnableServoAck )
   END_RUNG wire#w5
   RUNG wire#w5
      Contact( "Unit1.Em3.ControlNodes".cmUnwinderVirtualAxis.monitoring.statusWord1.Error )
   END_RUNG wire#w6
   RUNG wire#w6
      I_Contact( "Unit1.Em3.ControlNodes".cmUnwinderVirtualAxis.commands.enableAxis )
      Coil( "Unit1.Em3.ControlNodes".cmUnwinderVirtualAxis.commandConfiguration.generalSettings.resetWithRestart )
   END_RUNG
   // the same network as SCL:
   "Unit1.Em3.ControlNodes".cmCompensatorAxisX.commands.resetAxis := "Unit1.EmNodes".unitStatus.safetyReleased AND (#statUnitStatus.acknowledgeActive OR #statUnitStatus.state.resetting OR "Unit1.EmNodes".EnableServoAck) AND ("Unit1.Em3.ControlNodes".cmCompensatorAxisX.monitoring.error OR "Unit1.Em3.ControlNodes".cmCompensatorAxisX.monitoring.statusWord1.Error);
   "Unit1.Em3.ControlNodes".cmCompensatorAxisX.commandConfiguration.generalSettings.resetWithRestart := "Unit1.Em3.ControlNodes".cmCompensatorAxisX.commands.resetAxis AND NOT "Unit1.Em3.ControlNodes".cmCompensatorAxisX.commands.enableAxis;
   "Unit1.Em3.ControlNodes".cmUnwinderVirtualAxis.commands.resetAxis := "Unit1.EmNodes".unitStatus.safetyReleased AND (#statUnitStatus.acknowledgeActive OR #statUnitStatus.state.resetting OR "Unit1.EmNodes".EnableServoAck) AND ("Unit1.Em3.ControlNodes".cmUnwinderVirtualAxis.monitoring.error OR "Unit1.Em3.ControlNodes".cmUnwinderVirtualAxis.monitoring.statusWord1.Error);
   "Unit1.Em3.ControlNodes".cmUnwinderVirtualAxis.commandConfiguration.generalSettings.resetWithRestart := "Unit1.Em3.ControlNodes".cmUnwinderVirtualAxis.commands.resetAxis AND NOT "Unit1.Em3.ControlNodes".cmUnwinderVirtualAxis.commands.enableAxis;
END_REGION

REGION Network 32: Enable/Disable CMs
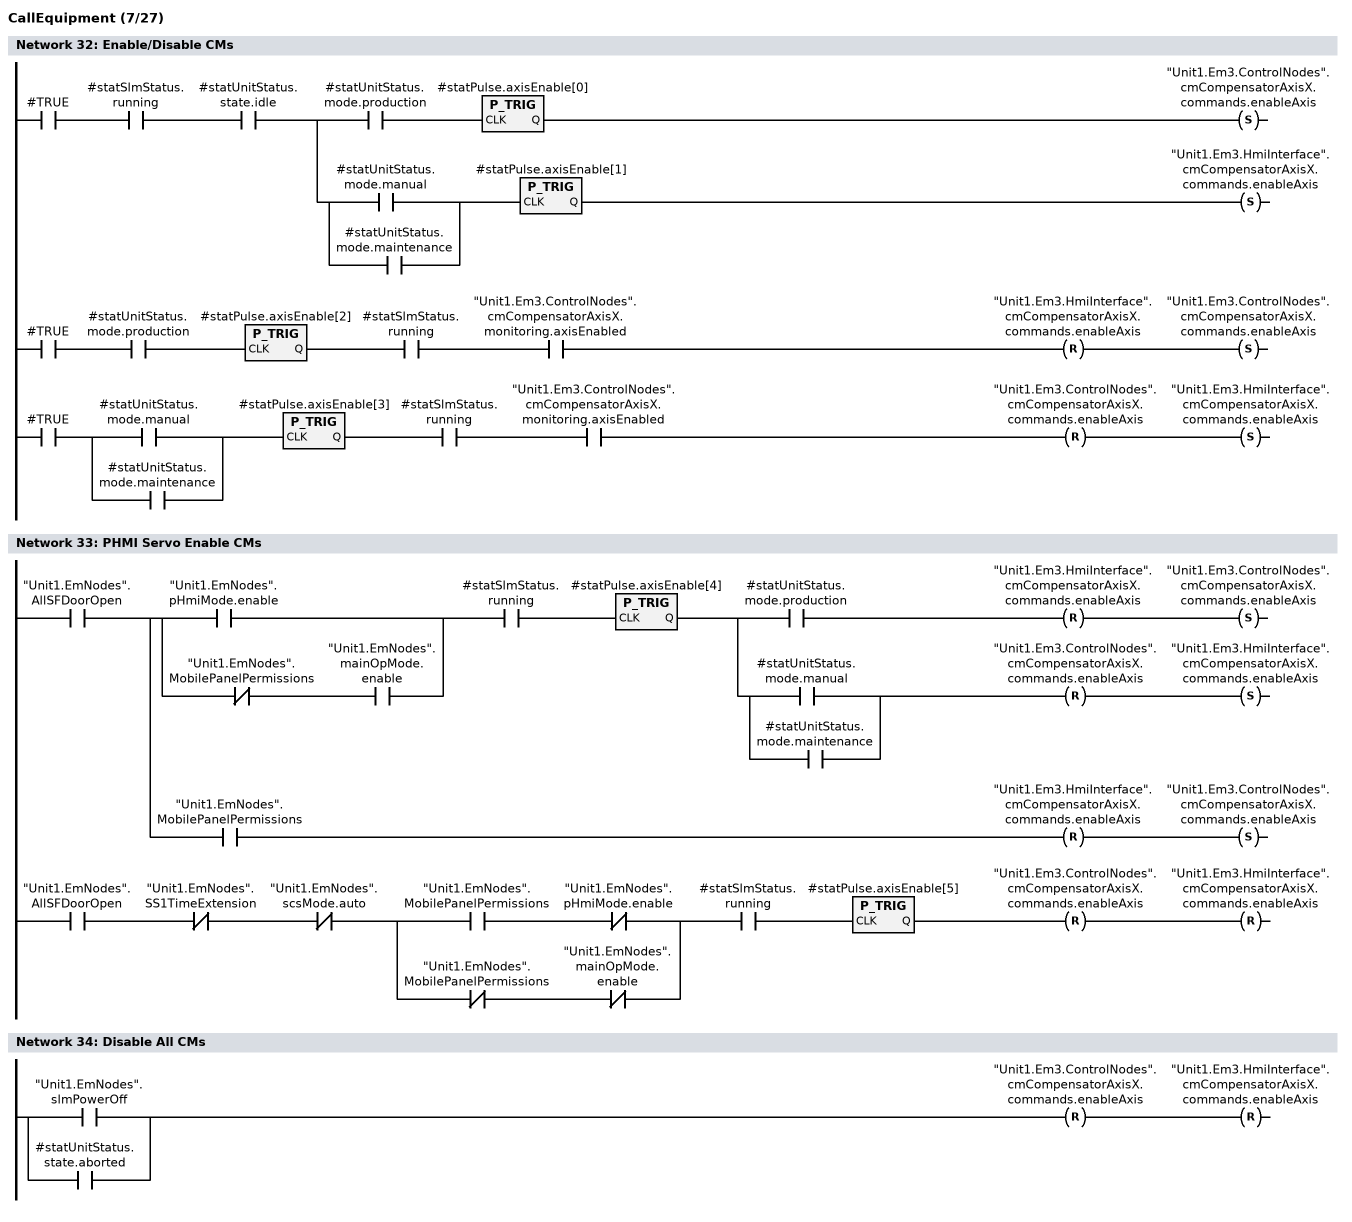
   RUNG wire#powerrail
      Contact( #TRUE )
      Contact( #statSlmStatus.running )
      Contact( #statUnitStatus.state.idle )
      wire#w1
      Contact( #statUnitStatus.mode.production )
      P_Trig( #statPulse.axisEnable[0] )
      S_Coil( "Unit1.Em3.ControlNodes".cmCompensatorAxisX.commands.enableAxis )
   END_RUNG
   RUNG wire#w1
      Contact( #statUnitStatus.mode.manual )
      wire#w2
      P_Trig( #statPulse.axisEnable[1] )
      S_Coil( "Unit1.Em3.HmiInterface".cmCompensatorAxisX.commands.enableAxis )
   END_RUNG
   RUNG wire#w1
      Contact( #statUnitStatus.mode.maintenance )
   END_RUNG wire#w2
   RUNG wire#powerrail
      Contact( #TRUE )
      Contact( #statUnitStatus.mode.production )
      P_Trig( #statPulse.axisEnable[2] )
      Contact( #statSlmStatus.running )
      Contact( "Unit1.Em3.ControlNodes".cmCompensatorAxisX.monitoring.axisEnabled )
      R_Coil( "Unit1.Em3.HmiInterface".cmCompensatorAxisX.commands.enableAxis )
      S_Coil( "Unit1.Em3.ControlNodes".cmCompensatorAxisX.commands.enableAxis )
   END_RUNG
   RUNG wire#powerrail
      Contact( #TRUE )
      wire#w3
      Contact( #statUnitStatus.mode.manual )
      wire#w4
      P_Trig( #statPulse.axisEnable[3] )
      Contact( #statSlmStatus.running )
      Contact( "Unit1.Em3.ControlNodes".cmCompensatorAxisX.monitoring.axisEnabled )
      R_Coil( "Unit1.Em3.ControlNodes".cmCompensatorAxisX.commands.enableAxis )
      S_Coil( "Unit1.Em3.HmiInterface".cmCompensatorAxisX.commands.enableAxis )
   END_RUNG
   RUNG wire#w3
      Contact( #statUnitStatus.mode.maintenance )
   END_RUNG wire#w4
   // the same network as SCL:
   #_w1 := #TRUE AND #statSlmStatus.running AND #statUnitStatus.state.idle;
   #_w2 := #_w1 AND #statUnitStatus.mode.production;
   #_w3 := #_w2 AND NOT #statPulse.axisEnable[0];   // rising edge
   #statPulse.axisEnable[0] := #_w2;
   IF #_w3 THEN "Unit1.Em3.ControlNodes".cmCompensatorAxisX.commands.enableAxis := TRUE; END_IF;
   #_w4 := #_w1 AND (#statUnitStatus.mode.manual OR #statUnitStatus.mode.maintenance);
   #_w5 := #_w4 AND NOT #statPulse.axisEnable[1];   // rising edge
   #statPulse.axisEnable[1] := #_w4;
   IF #_w5 THEN "Unit1.Em3.HmiInterface".cmCompensatorAxisX.commands.enableAxis := TRUE; END_IF;
   #_w6 := #TRUE AND #statUnitStatus.mode.production;
   #_w7 := #_w6 AND NOT #statPulse.axisEnable[2];   // rising edge
   #statPulse.axisEnable[2] := #_w6;
   IF #_w7 AND #statSlmStatus.running AND "Unit1.Em3.ControlNodes".cmCompensatorAxisX.monitoring.axisEnabled THEN
       "Unit1.Em3.HmiInterface".cmCompensatorAxisX.commands.enableAxis := FALSE;
       "Unit1.Em3.ControlNodes".cmCompensatorAxisX.commands.enableAxis := TRUE;
   END_IF;
   #_w8 := #TRUE AND (#statUnitStatus.mode.manual OR #statUnitStatus.mode.maintenance);
   #_w9 := #_w8 AND NOT #statPulse.axisEnable[3];   // rising edge
   #statPulse.axisEnable[3] := #_w8;
   IF #_w9 AND #statSlmStatus.running AND "Unit1.Em3.ControlNodes".cmCompensatorAxisX.monitoring.axisEnabled THEN
       "Unit1.Em3.ControlNodes".cmCompensatorAxisX.commands.enableAxis := FALSE;
       "Unit1.Em3.HmiInterface".cmCompensatorAxisX.commands.enableAxis := TRUE;
   END_IF;
END_REGION

REGION Network 33: PHMI Servo Enable CMs
   RUNG wire#powerrail
      Contact( "Unit1.EmNodes".AllSFDoorOpen )
      wire#w1
      Contact( "Unit1.EmNodes".pHmiMode.enable )
      wire#w2
      Contact( #statSlmStatus.running )
      P_Trig( #statPulse.axisEnable[4] )
      wire#w3
      Contact( #statUnitStatus.mode.production )
      R_Coil( "Unit1.Em3.HmiInterface".cmCompensatorAxisX.commands.enableAxis )
      S_Coil( "Unit1.Em3.ControlNodes".cmCompensatorAxisX.commands.enableAxis )
   END_RUNG
   RUNG wire#w1
      I_Contact( "Unit1.EmNodes".MobilePanelPermissions )
      Contact( "Unit1.EmNodes".mainOpMode.enable )
   END_RUNG wire#w2
   RUNG wire#w3
      Contact( #statUnitStatus.mode.manual )
      wire#w4
      R_Coil( "Unit1.Em3.ControlNodes".cmCompensatorAxisX.commands.enableAxis )
      S_Coil( "Unit1.Em3.HmiInterface".cmCompensatorAxisX.commands.enableAxis )
   END_RUNG
   RUNG wire#w3
      Contact( #statUnitStatus.mode.maintenance )
   END_RUNG wire#w4
   RUNG wire#w1
      Contact( "Unit1.EmNodes".MobilePanelPermissions )
      R_Coil( "Unit1.Em3.HmiInterface".cmCompensatorAxisX.commands.enableAxis )
      S_Coil( "Unit1.Em3.ControlNodes".cmCompensatorAxisX.commands.enableAxis )
   END_RUNG
   RUNG wire#powerrail
      Contact( "Unit1.EmNodes".AllSFDoorOpen )
      I_Contact( "Unit1.EmNodes".SS1TimeExtension )
      I_Contact( "Unit1.EmNodes".scsMode.auto )
      wire#w5
      Contact( "Unit1.EmNodes".MobilePanelPermissions )
      I_Contact( "Unit1.EmNodes".pHmiMode.enable )
      wire#w6
      Contact( #statSlmStatus.running )
      P_Trig( #statPulse.axisEnable[5] )
      R_Coil( "Unit1.Em3.ControlNodes".cmCompensatorAxisX.commands.enableAxis )
      R_Coil( "Unit1.Em3.HmiInterface".cmCompensatorAxisX.commands.enableAxis )
   END_RUNG
   RUNG wire#w5
      I_Contact( "Unit1.EmNodes".MobilePanelPermissions )
      I_Contact( "Unit1.EmNodes".mainOpMode.enable )
   END_RUNG wire#w6
   // the same network as SCL:
   #_w1 := "Unit1.EmNodes".AllSFDoorOpen AND ("Unit1.EmNodes".pHmiMode.enable OR (NOT "Unit1.EmNodes".MobilePanelPermissions AND "Unit1.EmNodes".mainOpMode.enable)) AND #statSlmStatus.running;
   #_w2 := #_w1 AND NOT #statPulse.axisEnable[4];   // rising edge
   #statPulse.axisEnable[4] := #_w1;
   IF #_w2 AND #statUnitStatus.mode.production THEN
       "Unit1.Em3.HmiInterface".cmCompensatorAxisX.commands.enableAxis := FALSE;
       "Unit1.Em3.ControlNodes".cmCompensatorAxisX.commands.enableAxis := TRUE;
   END_IF;
   IF #_w2 AND (#statUnitStatus.mode.manual OR #statUnitStatus.mode.maintenance) THEN
       "Unit1.Em3.ControlNodes".cmCompensatorAxisX.commands.enableAxis := FALSE;
       "Unit1.Em3.HmiInterface".cmCompensatorAxisX.commands.enableAxis := TRUE;
   END_IF;
   IF "Unit1.EmNodes".AllSFDoorOpen AND "Unit1.EmNodes".MobilePanelPermissions THEN
       "Unit1.Em3.HmiInterface".cmCompensatorAxisX.commands.enableAxis := FALSE;
       "Unit1.Em3.ControlNodes".cmCompensatorAxisX.commands.enableAxis := TRUE;
   END_IF;
   #_w3 := "Unit1.EmNodes".AllSFDoorOpen AND NOT "Unit1.EmNodes".SS1TimeExtension AND NOT "Unit1.EmNodes".scsMode.auto AND (("Unit1.EmNodes".MobilePanelPermissions AND NOT "Unit1.EmNodes".pHmiMode.enable) OR (NOT "Unit1.EmNodes".MobilePanelPermissions AND NOT "Unit1.EmNodes".mainOpMode.enable)) AND #statSlmStatus.running;
   #_w4 := #_w3 AND NOT #statPulse.axisEnable[5];   // rising edge
   #statPulse.axisEnable[5] := #_w3;
   IF #_w4 THEN
       "Unit1.Em3.ControlNodes".cmCompensatorAxisX.commands.enableAxis := FALSE;
       "Unit1.Em3.HmiInterface".cmCompensatorAxisX.commands.enableAxis := FALSE;
   END_IF;
END_REGION

REGION Network 34: Disable All CMs
   RUNG wire#powerrail
      Contact( "Unit1.EmNodes".slmPowerOff )
      wire#w1
      R_Coil( "Unit1.Em3.ControlNodes".cmCompensatorAxisX.commands.enableAxis )
      R_Coil( "Unit1.Em3.HmiInterface".cmCompensatorAxisX.commands.enableAxis )
   END_RUNG
   RUNG wire#powerrail
      Contact( #statUnitStatus.state.aborted )
   END_RUNG wire#w1
   // the same network as SCL:
   IF "Unit1.EmNodes".slmPowerOff OR #statUnitStatus.state.aborted THEN
       "Unit1.Em3.ControlNodes".cmCompensatorAxisX.commands.enableAxis := FALSE;
       "Unit1.Em3.HmiInterface".cmCompensatorAxisX.commands.enableAxis := FALSE;
   END_IF;
END_REGION

REGION Network 36: Unwinder Virtual Axis Enable
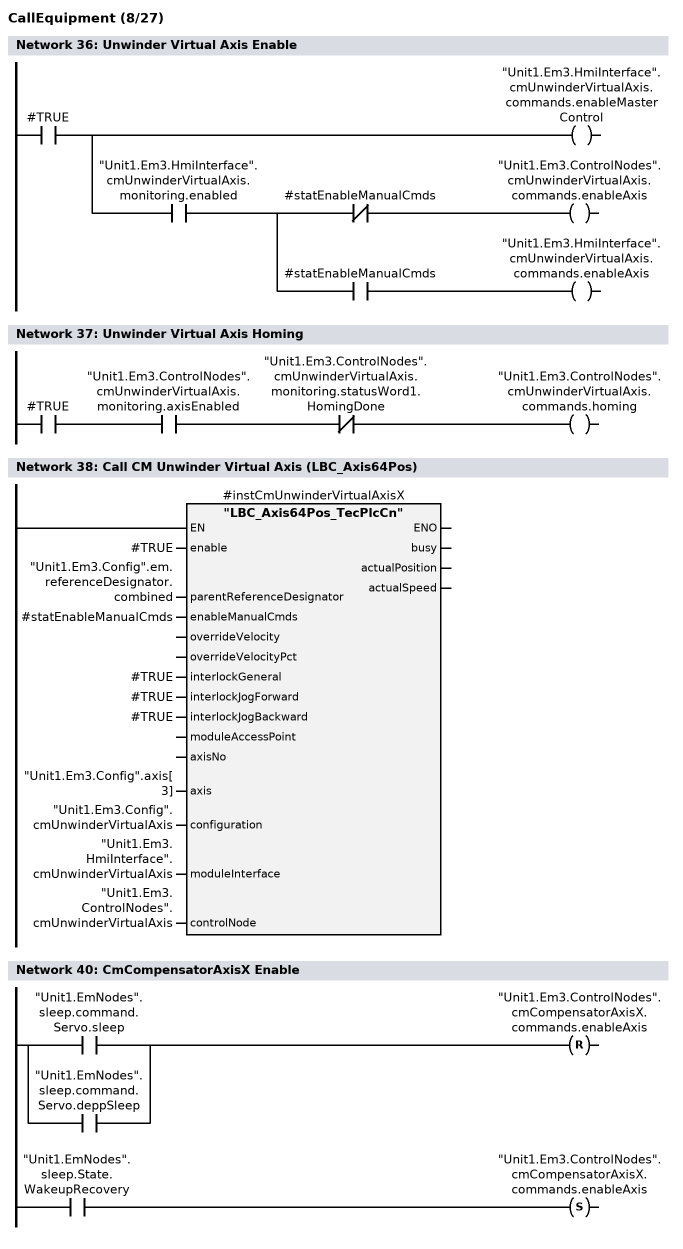
   RUNG wire#powerrail
      Contact( #TRUE )
      wire#w1
      Coil( "Unit1.Em3.HmiInterface".cmUnwinderVirtualAxis.commands.enableMasterControl )
   END_RUNG
   RUNG wire#w1
      Contact( "Unit1.Em3.HmiInterface".cmUnwinderVirtualAxis.monitoring.enabled )
      wire#w2
      I_Contact( #statEnableManualCmds )
      Coil( "Unit1.Em3.ControlNodes".cmUnwinderVirtualAxis.commands.enableAxis )
   END_RUNG
   RUNG wire#w2
      Contact( #statEnableManualCmds )
      Coil( "Unit1.Em3.HmiInterface".cmUnwinderVirtualAxis.commands.enableAxis )
   END_RUNG
   // the same network as SCL:
   "Unit1.Em3.HmiInterface".cmUnwinderVirtualAxis.commands.enableMasterControl := #TRUE;
   #_w1 := #TRUE AND "Unit1.Em3.HmiInterface".cmUnwinderVirtualAxis.monitoring.enabled;
   "Unit1.Em3.ControlNodes".cmUnwinderVirtualAxis.commands.enableAxis := #_w1 AND NOT #statEnableManualCmds;
   "Unit1.Em3.HmiInterface".cmUnwinderVirtualAxis.commands.enableAxis := #_w1 AND #statEnableManualCmds;
END_REGION

REGION Network 37: Unwinder Virtual Axis Homing
   RUNG wire#powerrail
      Contact( #TRUE )
      Contact( "Unit1.Em3.ControlNodes".cmUnwinderVirtualAxis.monitoring.axisEnabled )
      I_Contact( "Unit1.Em3.ControlNodes".cmUnwinderVirtualAxis.monitoring.statusWord1.HomingDone )
      Coil( "Unit1.Em3.ControlNodes".cmUnwinderVirtualAxis.commands.homing )
   END_RUNG
   // the same network as SCL:
   "Unit1.Em3.ControlNodes".cmUnwinderVirtualAxis.commands.homing := #TRUE AND "Unit1.Em3.ControlNodes".cmUnwinderVirtualAxis.monitoring.axisEnabled AND NOT "Unit1.Em3.ControlNodes".cmUnwinderVirtualAxis.monitoring.statusWord1.HomingDone;
END_REGION

REGION Network 38: Call CM Unwinder Virtual Axis (LBC_Axis64Pos)
   RUNG wire#powerrail
      #instCmUnwinderVirtualAxisX(enable := #TRUE, parentReferenceDesignator := "Unit1.Em3.Config".em.referenceDesignator.combined, enableManualCmds := #statEnableManualCmds, overrideVelocity :=, overrideVelocityPct :=, interlockGeneral := #TRUE, interlockJogForward := #TRUE, interlockJogBackward := #TRUE, moduleAccessPoint :=, axisNo :=, axis := "Unit1.Em3.Config".axis[3], configuration := "Unit1.Em3.Config".cmUnwinderVirtualAxis, moduleInterface := "Unit1.Em3.HmiInterface".cmUnwinderVirtualAxis, controlNode := "Unit1.Em3.ControlNodes".cmUnwinderVirtualAxis, busy =>, actualPosition =>, actualSpeed =>)
   END_RUNG
   // the same network as SCL:
   #instCmUnwinderVirtualAxisX(enable := #TRUE,   // "LBC_Axis64Pos_TecPlcCn"
                           parentReferenceDesignator := "Unit1.Em3.Config".em.referenceDesignator.combined,
                           enableManualCmds := #statEnableManualCmds,
                           interlockGeneral := #TRUE,
                           interlockJogForward := #TRUE,
                           interlockJogBackward := #TRUE,
                           axis := "Unit1.Em3.Config".axis[3],
                           configuration := "Unit1.Em3.Config".cmUnwinderVirtualAxis,
                           moduleInterface := "Unit1.Em3.HmiInterface".cmUnwinderVirtualAxis,
                           controlNode := "Unit1.Em3.ControlNodes".cmUnwinderVirtualAxis);
END_REGION

REGION Network 40: CmCompensatorAxisX Enable
   RUNG wire#powerrail
      Contact( "Unit1.EmNodes".sleep.command.Servo.sleep )
      wire#w1
      R_Coil( "Unit1.Em3.ControlNodes".cmCompensatorAxisX.commands.enableAxis )
   END_RUNG
   RUNG wire#powerrail
      Contact( "Unit1.EmNodes".sleep.command.Servo.deppSleep )
   END_RUNG wire#w1
   RUNG wire#powerrail
      Contact( "Unit1.EmNodes".sleep.State.WakeupRecovery )
      S_Coil( "Unit1.Em3.ControlNodes".cmCompensatorAxisX.commands.enableAxis )
   END_RUNG
   // the same network as SCL:
   IF "Unit1.EmNodes".sleep.command.Servo.sleep OR "Unit1.EmNodes".sleep.command.Servo.deppSleep THEN
       "Unit1.Em3.ControlNodes".cmCompensatorAxisX.commands.enableAxis := FALSE;
   END_IF;
   IF "Unit1.EmNodes".sleep.State.WakeupRecovery THEN
       "Unit1.Em3.ControlNodes".cmCompensatorAxisX.commands.enableAxis := TRUE;
   END_IF;
END_REGION

REGION Network 41: Interlock/Servo
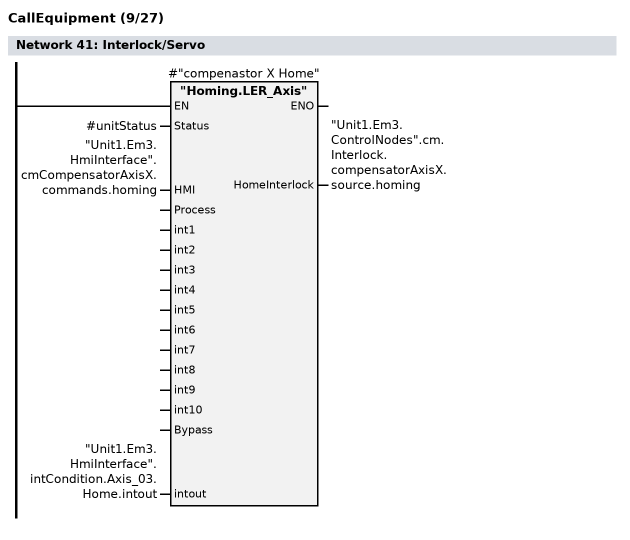
   RUNG wire#powerrail
      #"compenastor X Home"(Status := #unitStatus, HMI := "Unit1.Em3.HmiInterface".cmCompensatorAxisX.commands.homing, Process :=, int1 :=, int2 :=, int3 :=, int4 :=, int5 :=, int6 :=, int7 :=, int8 :=, int9 :=, int10 :=, Bypass :=, intout := "Unit1.Em3.HmiInterface".intCondition.Axis_03.Home.intout, HomeInterlock => "Unit1.Em3.ControlNodes".cm.Interlock.compensatorAxisX.source.homing)
   END_RUNG
   // the same network as SCL:
   #"compenastor X Home"(Status := #unitStatus,   // "Homing.LER_Axis"
                         HMI := "Unit1.Em3.HmiInterface".cmCompensatorAxisX.commands.homing,
                         intout := "Unit1.Em3.HmiInterface".intCondition.Axis_03.Home.intout,
                         HomeInterlock => "Unit1.Em3.ControlNodes".cm.Interlock.compensatorAxisX.source.homing);
END_REGION

REGION Network 42: CmCompensatorAxisX Position Absolute Jog
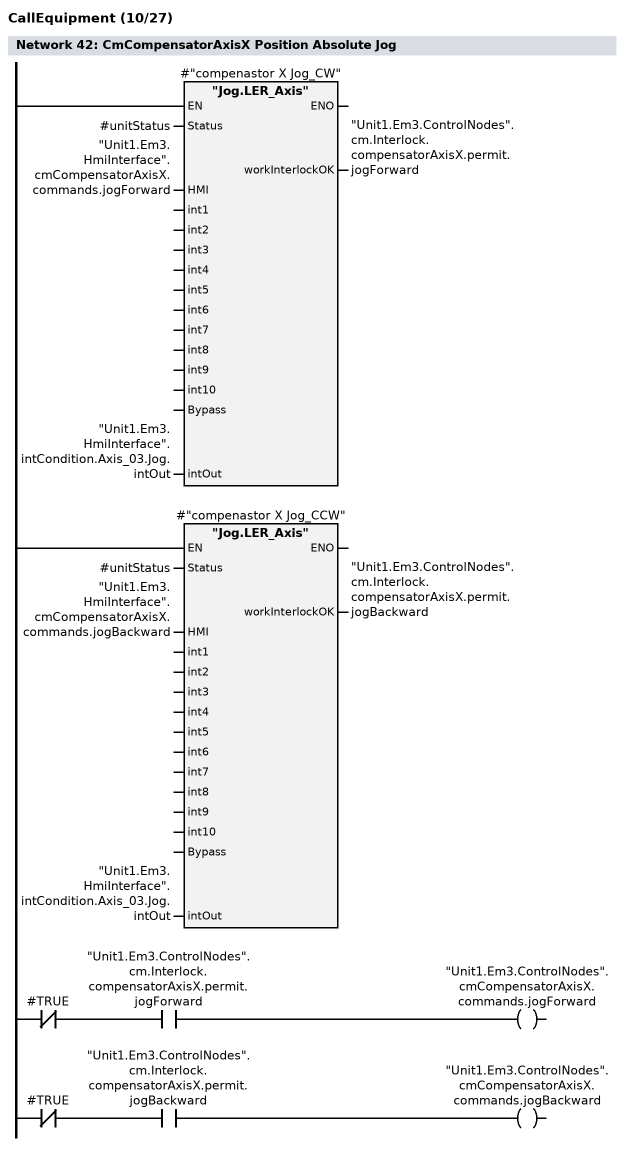
   RUNG wire#powerrail
      #"compenastor X Jog_CW"(Status := #unitStatus, HMI := "Unit1.Em3.HmiInterface".cmCompensatorAxisX.commands.jogForward, int1 :=, int2 :=, int3 :=, int4 :=, int5 :=, int6 :=, int7 :=, int8 :=, int9 :=, int10 :=, Bypass :=, intOut := "Unit1.Em3.HmiInterface".intCondition.Axis_03.Jog.intOut, workInterlockOK => "Unit1.Em3.ControlNodes".cm.Interlock.compensatorAxisX.permit.jogForward)
   END_RUNG
   RUNG wire#powerrail
      #"compenastor X Jog_CCW"(Status := #unitStatus, HMI := "Unit1.Em3.HmiInterface".cmCompensatorAxisX.commands.jogBackward, int1 :=, int2 :=, int3 :=, int4 :=, int5 :=, int6 :=, int7 :=, int8 :=, int9 :=, int10 :=, Bypass :=, intOut := "Unit1.Em3.HmiInterface".intCondition.Axis_03.Jog.intOut, workInterlockOK => "Unit1.Em3.ControlNodes".cm.Interlock.compensatorAxisX.permit.jogBackward)
   END_RUNG
   RUNG wire#powerrail
      I_Contact( #TRUE )
      Contact( "Unit1.Em3.ControlNodes".cm.Interlock.compensatorAxisX.permit.jogForward )
      Coil( "Unit1.Em3.ControlNodes".cmCompensatorAxisX.commands.jogForward )
   END_RUNG
   RUNG wire#powerrail
      I_Contact( #TRUE )
      Contact( "Unit1.Em3.ControlNodes".cm.Interlock.compensatorAxisX.permit.jogBackward )
      Coil( "Unit1.Em3.ControlNodes".cmCompensatorAxisX.commands.jogBackward )
   END_RUNG
   // the same network as SCL:
   #"compenastor X Jog_CW"(Status := #unitStatus,   // "Jog.LER_Axis"
                           HMI := "Unit1.Em3.HmiInterface".cmCompensatorAxisX.commands.jogForward,
                           intOut := "Unit1.Em3.HmiInterface".intCondition.Axis_03.Jog.intOut,
                           workInterlockOK => "Unit1.Em3.ControlNodes".cm.Interlock.compensatorAxisX.permit.jogForward);
   #"compenastor X Jog_CCW"(Status := #unitStatus,   // "Jog.LER_Axis"
                           HMI := "Unit1.Em3.HmiInterface".cmCompensatorAxisX.commands.jogBackward,
                           intOut := "Unit1.Em3.HmiInterface".intCondition.Axis_03.Jog.intOut,
                           workInterlockOK => "Unit1.Em3.ControlNodes".cm.Interlock.compensatorAxisX.permit.jogBackward);
   "Unit1.Em3.ControlNodes".cmCompensatorAxisX.commands.jogForward := NOT #TRUE AND "Unit1.Em3.ControlNodes".cm.Interlock.compensatorAxisX.permit.jogForward;
   "Unit1.Em3.ControlNodes".cmCompensatorAxisX.commands.jogBackward := NOT #TRUE AND "Unit1.Em3.ControlNodes".cm.Interlock.compensatorAxisX.permit.jogBackward;
END_REGION

REGION Network 43: CmCompensatorAxisX Position Absolute Position0
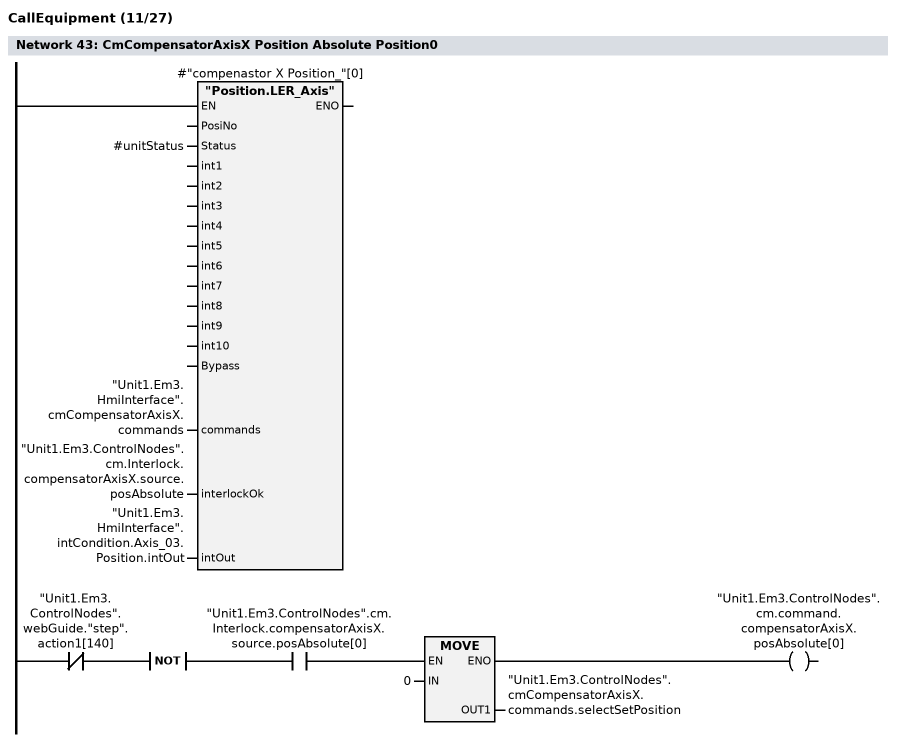
   RUNG wire#powerrail
      #"compenastor X Position_"[0](PosiNo :=, Status := #unitStatus, int1 :=, int2 :=, int3 :=, int4 :=, int5 :=, int6 :=, int7 :=, int8 :=, int9 :=, int10 :=, Bypass :=, commands := "Unit1.Em3.HmiInterface".cmCompensatorAxisX.commands, interlockOk := "Unit1.Em3.ControlNodes".cm.Interlock.compensatorAxisX.source.posAbsolute, intOut := "Unit1.Em3.HmiInterface".intCondition.Axis_03.Position.intOut)
   END_RUNG
   RUNG wire#powerrail
      I_Contact( "Unit1.Em3.ControlNodes".webGuide."step".action1[140] )
      Not()
      Contact( "Unit1.Em3.ControlNodes".cm.Interlock.compensatorAxisX.source.posAbsolute[0] )
      Move(in := 0, out1 => "Unit1.Em3.ControlNodes".cmCompensatorAxisX.commands.selectSetPosition)
      Coil( "Unit1.Em3.ControlNodes".cm.command.compensatorAxisX.posAbsolute[0] )
   END_RUNG
   // the same network as SCL:
   #"compenastor X Position_"[0](Status := #unitStatus,   // "Position.LER_Axis"
                           commands := "Unit1.Em3.HmiInterface".cmCompensatorAxisX.commands,
                           interlockOk := "Unit1.Em3.ControlNodes".cm.Interlock.compensatorAxisX.source.posAbsolute,
                           intOut := "Unit1.Em3.HmiInterface".intCondition.Axis_03.Position.intOut);
   #_w1 := NOT (NOT "Unit1.Em3.ControlNodes".webGuide."step".action1[140]) AND "Unit1.Em3.ControlNodes".cm.Interlock.compensatorAxisX.source.posAbsolute[0];
   IF #_w1 THEN "Unit1.Em3.ControlNodes".cmCompensatorAxisX.commands.selectSetPosition := 0; END_IF;
   "Unit1.Em3.ControlNodes".cm.command.compensatorAxisX.posAbsolute[0] := #_w1;
END_REGION

REGION Network 44: CmCompensatorAxisX Position Absolute Position1
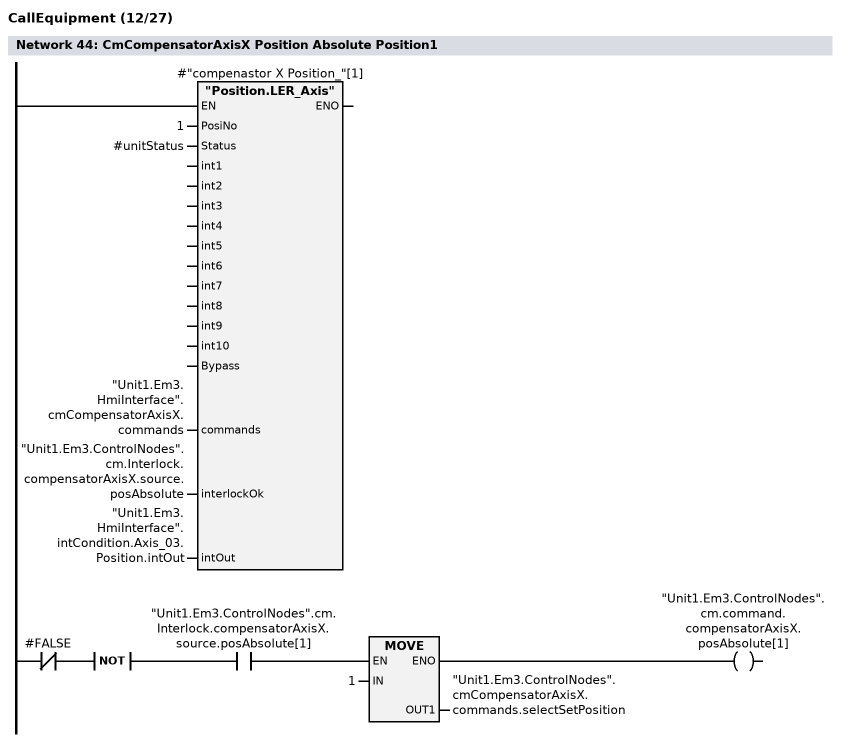
   RUNG wire#powerrail
      #"compenastor X Position_"[1](PosiNo := 1, Status := #unitStatus, int1 :=, int2 :=, int3 :=, int4 :=, int5 :=, int6 :=, int7 :=, int8 :=, int9 :=, int10 :=, Bypass :=, commands := "Unit1.Em3.HmiInterface".cmCompensatorAxisX.commands, interlockOk := "Unit1.Em3.ControlNodes".cm.Interlock.compensatorAxisX.source.posAbsolute, intOut := "Unit1.Em3.HmiInterface".intCondition.Axis_03.Position.intOut)
   END_RUNG
   RUNG wire#powerrail
      I_Contact( #FALSE )
      Not()
      Contact( "Unit1.Em3.ControlNodes".cm.Interlock.compensatorAxisX.source.posAbsolute[1] )
      Move(in := 1, out1 => "Unit1.Em3.ControlNodes".cmCompensatorAxisX.commands.selectSetPosition)
      Coil( "Unit1.Em3.ControlNodes".cm.command.compensatorAxisX.posAbsolute[1] )
   END_RUNG
   // the same network as SCL:
   #"compenastor X Position_"[1](PosiNo := 1,   // "Position.LER_Axis"
                           Status := #unitStatus,
                           commands := "Unit1.Em3.HmiInterface".cmCompensatorAxisX.commands,
                           interlockOk := "Unit1.Em3.ControlNodes".cm.Interlock.compensatorAxisX.source.posAbsolute,
                           intOut := "Unit1.Em3.HmiInterface".intCondition.Axis_03.Position.intOut);
   #_w1 := NOT (NOT #FALSE) AND "Unit1.Em3.ControlNodes".cm.Interlock.compensatorAxisX.source.posAbsolute[1];
   IF #_w1 THEN "Unit1.Em3.ControlNodes".cmCompensatorAxisX.commands.selectSetPosition := 1; END_IF;
   "Unit1.Em3.ControlNodes".cm.command.compensatorAxisX.posAbsolute[1] := #_w1;
END_REGION

REGION Network 45: CmCompensatorAxisX Position Absolute Position2
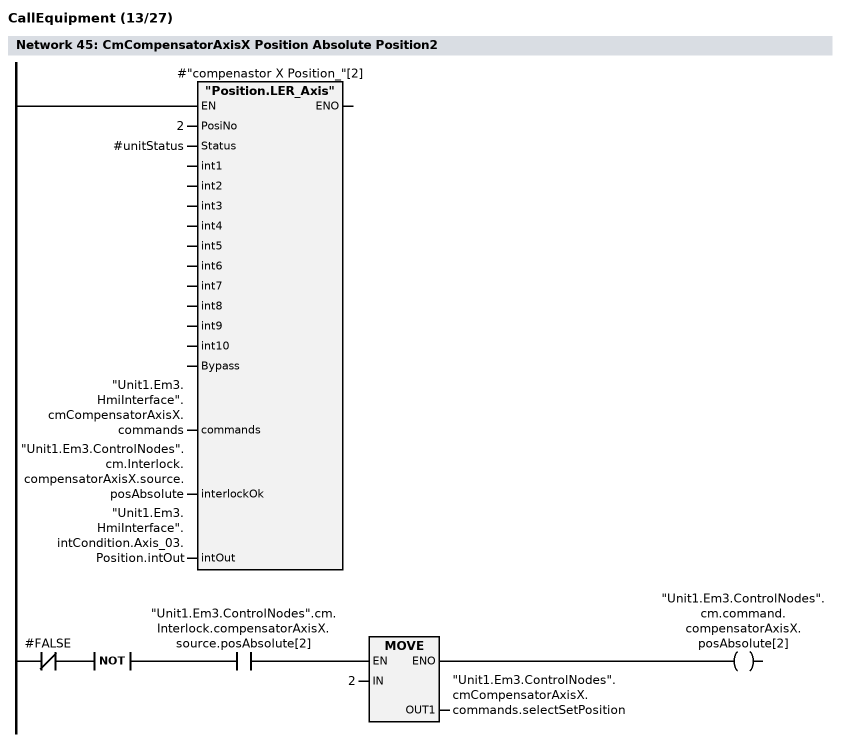
   RUNG wire#powerrail
      #"compenastor X Position_"[2](PosiNo := 2, Status := #unitStatus, int1 :=, int2 :=, int3 :=, int4 :=, int5 :=, int6 :=, int7 :=, int8 :=, int9 :=, int10 :=, Bypass :=, commands := "Unit1.Em3.HmiInterface".cmCompensatorAxisX.commands, interlockOk := "Unit1.Em3.ControlNodes".cm.Interlock.compensatorAxisX.source.posAbsolute, intOut := "Unit1.Em3.HmiInterface".intCondition.Axis_03.Position.intOut)
   END_RUNG
   RUNG wire#powerrail
      I_Contact( #FALSE )
      Not()
      Contact( "Unit1.Em3.ControlNodes".cm.Interlock.compensatorAxisX.source.posAbsolute[2] )
      Move(in := 2, out1 => "Unit1.Em3.ControlNodes".cmCompensatorAxisX.commands.selectSetPosition)
      Coil( "Unit1.Em3.ControlNodes".cm.command.compensatorAxisX.posAbsolute[2] )
   END_RUNG
   // the same network as SCL:
   #"compenastor X Position_"[2](PosiNo := 2,   // "Position.LER_Axis"
                           Status := #unitStatus,
                           commands := "Unit1.Em3.HmiInterface".cmCompensatorAxisX.commands,
                           interlockOk := "Unit1.Em3.ControlNodes".cm.Interlock.compensatorAxisX.source.posAbsolute,
                           intOut := "Unit1.Em3.HmiInterface".intCondition.Axis_03.Position.intOut);
   #_w1 := NOT (NOT #FALSE) AND "Unit1.Em3.ControlNodes".cm.Interlock.compensatorAxisX.source.posAbsolute[2];
   IF #_w1 THEN "Unit1.Em3.ControlNodes".cmCompensatorAxisX.commands.selectSetPosition := 2; END_IF;
   "Unit1.Em3.ControlNodes".cm.command.compensatorAxisX.posAbsolute[2] := #_w1;
END_REGION

REGION Network 46: CmCompensatorAxisX Position Absolute Position3
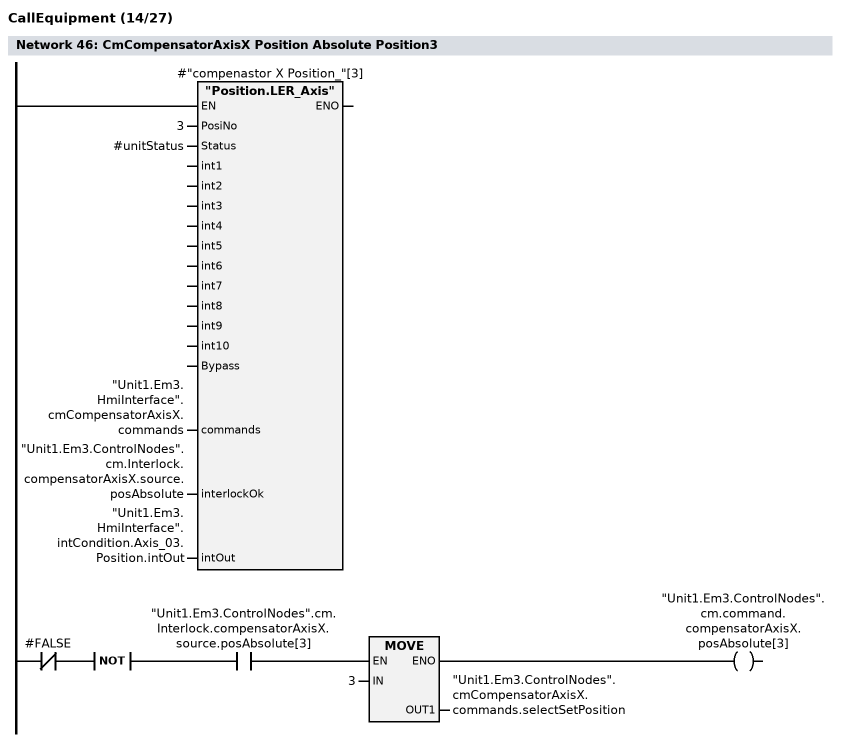
   RUNG wire#powerrail
      #"compenastor X Position_"[3](PosiNo := 3, Status := #unitStatus, int1 :=, int2 :=, int3 :=, int4 :=, int5 :=, int6 :=, int7 :=, int8 :=, int9 :=, int10 :=, Bypass :=, commands := "Unit1.Em3.HmiInterface".cmCompensatorAxisX.commands, interlockOk := "Unit1.Em3.ControlNodes".cm.Interlock.compensatorAxisX.source.posAbsolute, intOut := "Unit1.Em3.HmiInterface".intCondition.Axis_03.Position.intOut)
   END_RUNG
   RUNG wire#powerrail
      I_Contact( #FALSE )
      Not()
      Contact( "Unit1.Em3.ControlNodes".cm.Interlock.compensatorAxisX.source.posAbsolute[3] )
      Move(in := 3, out1 => "Unit1.Em3.ControlNodes".cmCompensatorAxisX.commands.selectSetPosition)
      Coil( "Unit1.Em3.ControlNodes".cm.command.compensatorAxisX.posAbsolute[3] )
   END_RUNG
   // the same network as SCL:
   #"compenastor X Position_"[3](PosiNo := 3,   // "Position.LER_Axis"
                           Status := #unitStatus,
                           commands := "Unit1.Em3.HmiInterface".cmCompensatorAxisX.commands,
                           interlockOk := "Unit1.Em3.ControlNodes".cm.Interlock.compensatorAxisX.source.posAbsolute,
                           intOut := "Unit1.Em3.HmiInterface".intCondition.Axis_03.Position.intOut);
   #_w1 := NOT (NOT #FALSE) AND "Unit1.Em3.ControlNodes".cm.Interlock.compensatorAxisX.source.posAbsolute[3];
   IF #_w1 THEN "Unit1.Em3.ControlNodes".cmCompensatorAxisX.commands.selectSetPosition := 3; END_IF;
   "Unit1.Em3.ControlNodes".cm.command.compensatorAxisX.posAbsolute[3] := #_w1;
END_REGION

REGION Network 47: CmCompensatorAxisX Position Absolute Position4
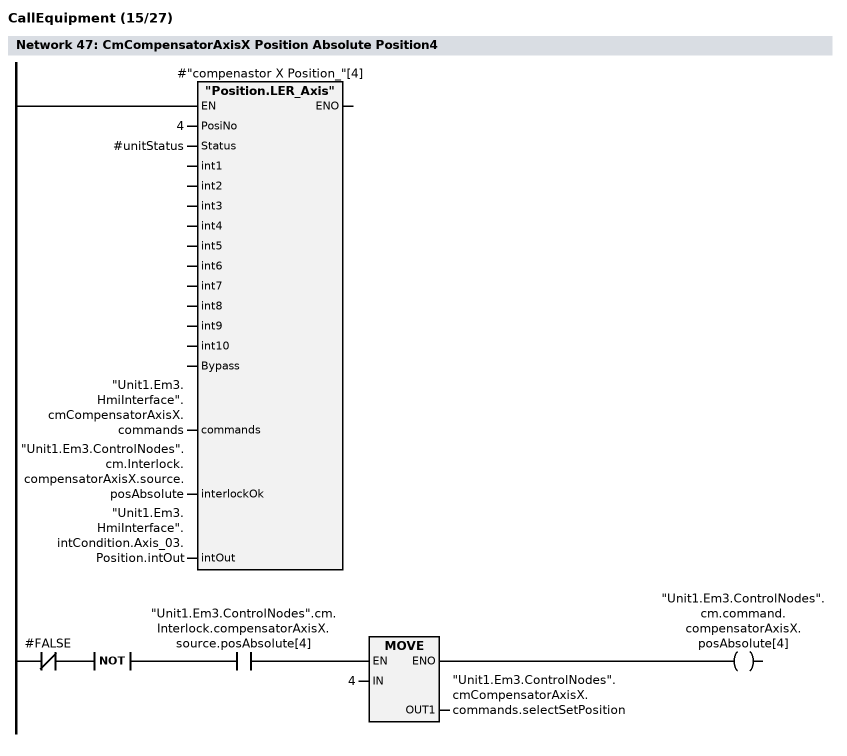
   RUNG wire#powerrail
      #"compenastor X Position_"[4](PosiNo := 4, Status := #unitStatus, int1 :=, int2 :=, int3 :=, int4 :=, int5 :=, int6 :=, int7 :=, int8 :=, int9 :=, int10 :=, Bypass :=, commands := "Unit1.Em3.HmiInterface".cmCompensatorAxisX.commands, interlockOk := "Unit1.Em3.ControlNodes".cm.Interlock.compensatorAxisX.source.posAbsolute, intOut := "Unit1.Em3.HmiInterface".intCondition.Axis_03.Position.intOut)
   END_RUNG
   RUNG wire#powerrail
      I_Contact( #FALSE )
      Not()
      Contact( "Unit1.Em3.ControlNodes".cm.Interlock.compensatorAxisX.source.posAbsolute[4] )
      Move(in := 4, out1 => "Unit1.Em3.ControlNodes".cmCompensatorAxisX.commands.selectSetPosition)
      Coil( "Unit1.Em3.ControlNodes".cm.command.compensatorAxisX.posAbsolute[4] )
   END_RUNG
   // the same network as SCL:
   #"compenastor X Position_"[4](PosiNo := 4,   // "Position.LER_Axis"
                           Status := #unitStatus,
                           commands := "Unit1.Em3.HmiInterface".cmCompensatorAxisX.commands,
                           interlockOk := "Unit1.Em3.ControlNodes".cm.Interlock.compensatorAxisX.source.posAbsolute,
                           intOut := "Unit1.Em3.HmiInterface".intCondition.Axis_03.Position.intOut);
   #_w1 := NOT (NOT #FALSE) AND "Unit1.Em3.ControlNodes".cm.Interlock.compensatorAxisX.source.posAbsolute[4];
   IF #_w1 THEN "Unit1.Em3.ControlNodes".cmCompensatorAxisX.commands.selectSetPosition := 4; END_IF;
   "Unit1.Em3.ControlNodes".cm.command.compensatorAxisX.posAbsolute[4] := #_w1;
END_REGION

REGION Network 48: CmCompensatorAxisX Position Absolute Position5
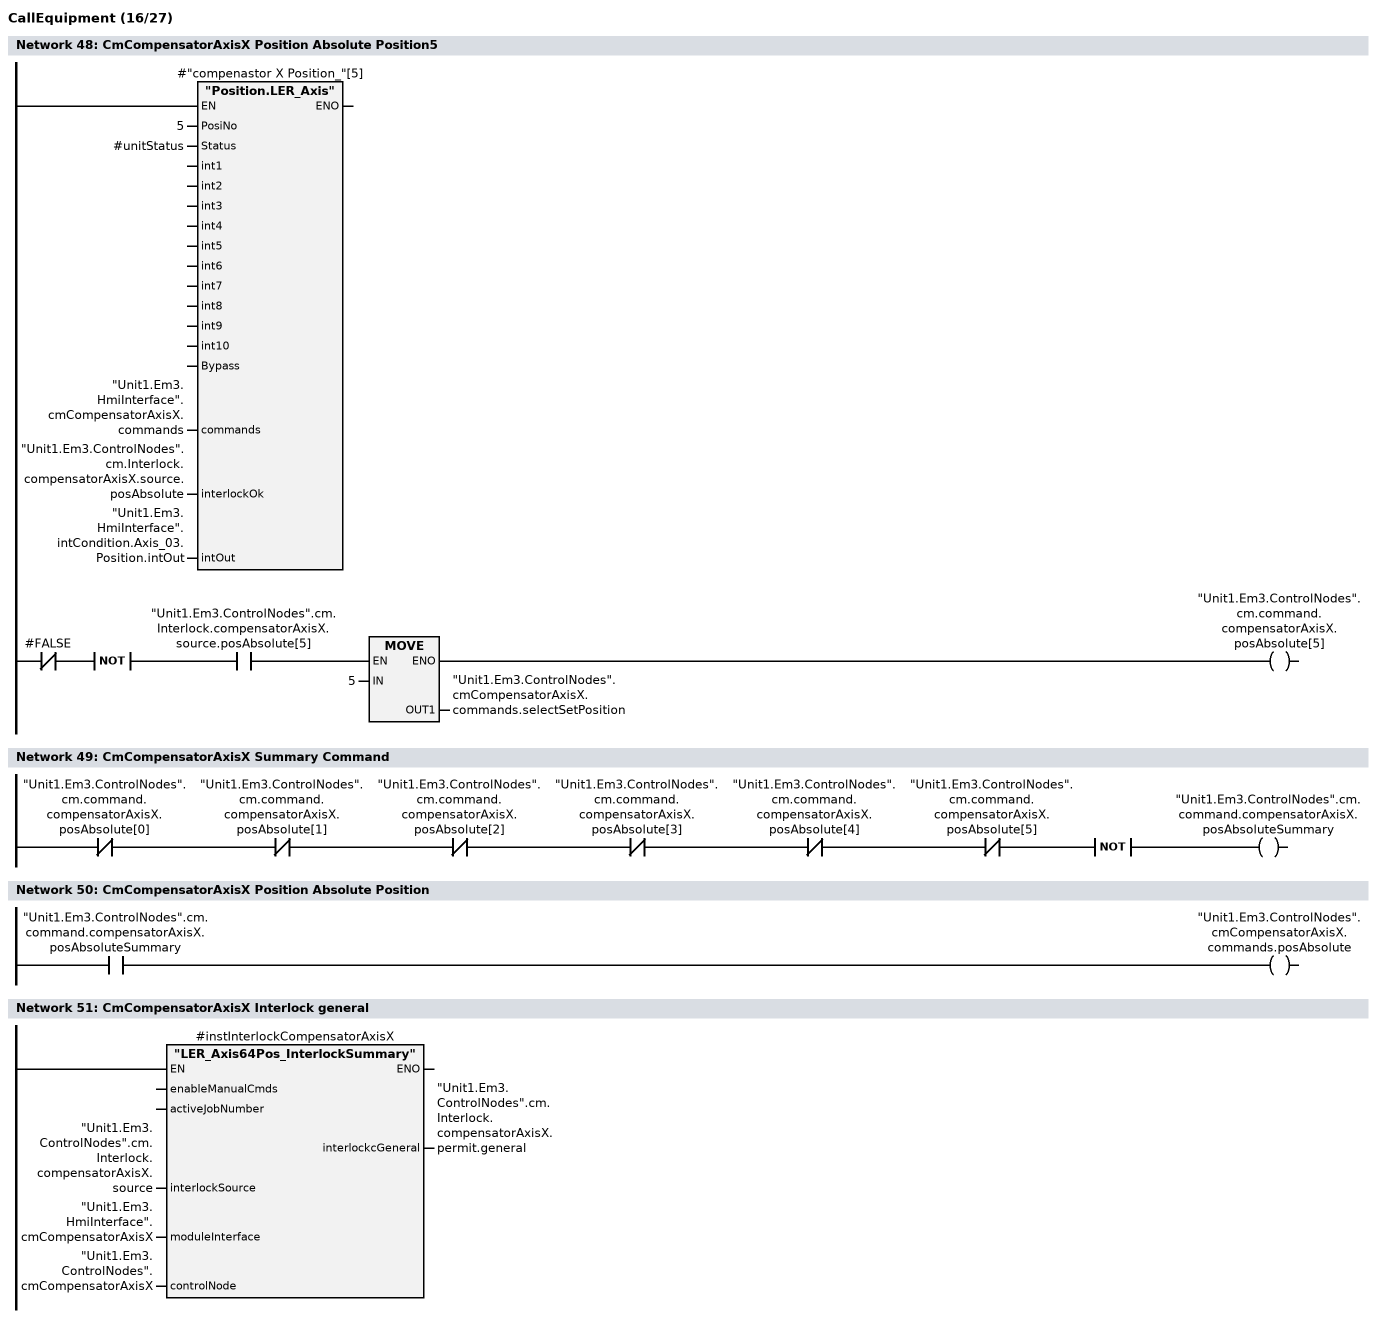
   RUNG wire#powerrail
      #"compenastor X Position_"[5](PosiNo := 5, Status := #unitStatus, int1 :=, int2 :=, int3 :=, int4 :=, int5 :=, int6 :=, int7 :=, int8 :=, int9 :=, int10 :=, Bypass :=, commands := "Unit1.Em3.HmiInterface".cmCompensatorAxisX.commands, interlockOk := "Unit1.Em3.ControlNodes".cm.Interlock.compensatorAxisX.source.posAbsolute, intOut := "Unit1.Em3.HmiInterface".intCondition.Axis_03.Position.intOut)
   END_RUNG
   RUNG wire#powerrail
      I_Contact( #FALSE )
      Not()
      Contact( "Unit1.Em3.ControlNodes".cm.Interlock.compensatorAxisX.source.posAbsolute[5] )
      Move(in := 5, out1 => "Unit1.Em3.ControlNodes".cmCompensatorAxisX.commands.selectSetPosition)
      Coil( "Unit1.Em3.ControlNodes".cm.command.compensatorAxisX.posAbsolute[5] )
   END_RUNG
   // the same network as SCL:
   #"compenastor X Position_"[5](PosiNo := 5,   // "Position.LER_Axis"
                           Status := #unitStatus,
                           commands := "Unit1.Em3.HmiInterface".cmCompensatorAxisX.commands,
                           interlockOk := "Unit1.Em3.ControlNodes".cm.Interlock.compensatorAxisX.source.posAbsolute,
                           intOut := "Unit1.Em3.HmiInterface".intCondition.Axis_03.Position.intOut);
   #_w1 := NOT (NOT #FALSE) AND "Unit1.Em3.ControlNodes".cm.Interlock.compensatorAxisX.source.posAbsolute[5];
   IF #_w1 THEN "Unit1.Em3.ControlNodes".cmCompensatorAxisX.commands.selectSetPosition := 5; END_IF;
   "Unit1.Em3.ControlNodes".cm.command.compensatorAxisX.posAbsolute[5] := #_w1;
END_REGION

REGION Network 49: CmCompensatorAxisX Summary Command
   RUNG wire#powerrail
      I_Contact( "Unit1.Em3.ControlNodes".cm.command.compensatorAxisX.posAbsolute[0] )
      I_Contact( "Unit1.Em3.ControlNodes".cm.command.compensatorAxisX.posAbsolute[1] )
      I_Contact( "Unit1.Em3.ControlNodes".cm.command.compensatorAxisX.posAbsolute[2] )
      I_Contact( "Unit1.Em3.ControlNodes".cm.command.compensatorAxisX.posAbsolute[3] )
      I_Contact( "Unit1.Em3.ControlNodes".cm.command.compensatorAxisX.posAbsolute[4] )
      I_Contact( "Unit1.Em3.ControlNodes".cm.command.compensatorAxisX.posAbsolute[5] )
      Not()
      Coil( "Unit1.Em3.ControlNodes".cm.command.compensatorAxisX.posAbsoluteSummary )
   END_RUNG
   // the same network as SCL:
   "Unit1.Em3.ControlNodes".cm.command.compensatorAxisX.posAbsoluteSummary := NOT (NOT "Unit1.Em3.ControlNodes".cm.command.compensatorAxisX.posAbsolute[0] AND NOT "Unit1.Em3.ControlNodes".cm.command.compensatorAxisX.posAbsolute[1] AND NOT "Unit1.Em3.ControlNodes".cm.command.compensatorAxisX.posAbsolute[2] AND NOT "Unit1.Em3.ControlNodes".cm.command.compensatorAxisX.posAbsolute[3] AND NOT "Unit1.Em3.ControlNodes".cm.command.compensatorAxisX.posAbsolute[4] AND NOT "Unit1.Em3.ControlNodes".cm.command.compensatorAxisX.posAbsolute[5]);
END_REGION

REGION Network 50: CmCompensatorAxisX Position Absolute Position
   RUNG wire#powerrail
      Contact( "Unit1.Em3.ControlNodes".cm.command.compensatorAxisX.posAbsoluteSummary )
      Coil( "Unit1.Em3.ControlNodes".cmCompensatorAxisX.commands.posAbsolute )
   END_RUNG
   // the same network as SCL:
   "Unit1.Em3.ControlNodes".cmCompensatorAxisX.commands.posAbsolute := "Unit1.Em3.ControlNodes".cm.command.compensatorAxisX.posAbsoluteSummary;
END_REGION

REGION Network 51: CmCompensatorAxisX Interlock general
   RUNG wire#powerrail
      #instInterlockCompensatorAxisX(enableManualCmds :=, activeJobNumber :=, interlockSource := "Unit1.Em3.ControlNodes".cm.Interlock.compensatorAxisX.source, moduleInterface := "Unit1.Em3.HmiInterface".cmCompensatorAxisX, controlNode := "Unit1.Em3.ControlNodes".cmCompensatorAxisX, interlockcGeneral => "Unit1.Em3.ControlNodes".cm.Interlock.compensatorAxisX.permit.general)
   END_RUNG
   // the same network as SCL:
   #instInterlockCompensatorAxisX(interlockSource := "Unit1.Em3.ControlNodes".cm.Interlock.compensatorAxisX.source,   // "LER_Axis64Pos_InterlockSummary"
                           moduleInterface := "Unit1.Em3.HmiInterface".cmCompensatorAxisX,
                           controlNode := "Unit1.Em3.ControlNodes".cmCompensatorAxisX,
                           interlockcGeneral => "Unit1.Em3.ControlNodes".cm.Interlock.compensatorAxisX.permit.general);
END_REGION

REGION Network 52: CmCompensatorAxisX velocity/speed
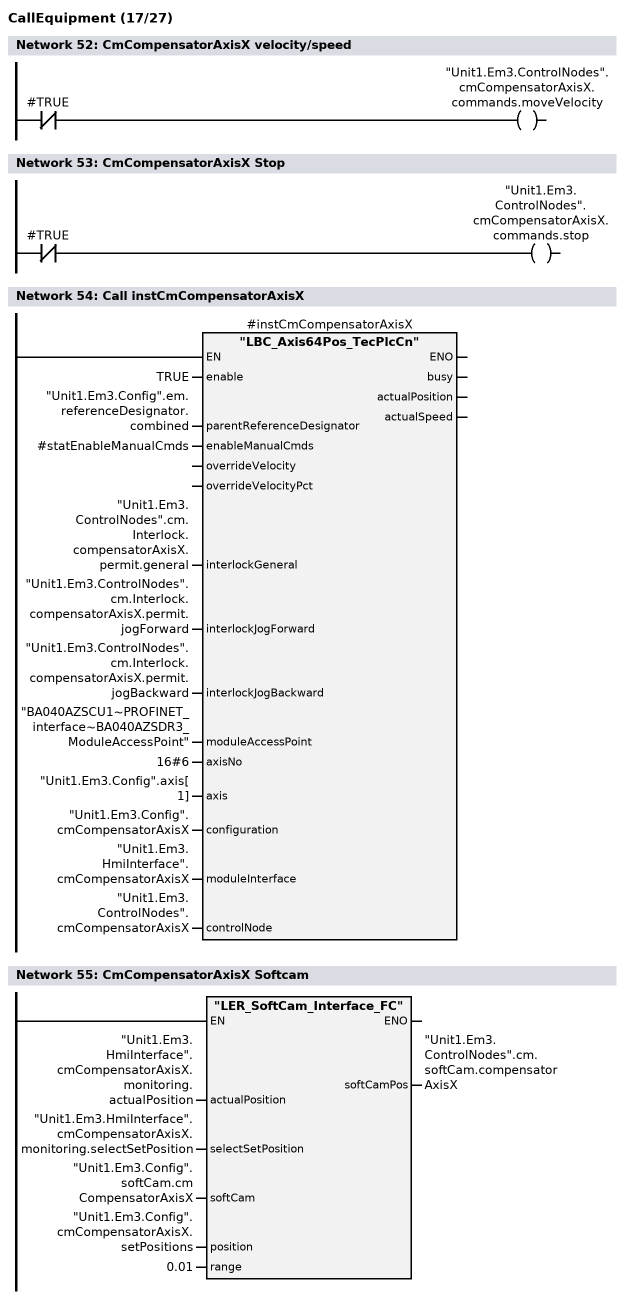
   RUNG wire#powerrail
      I_Contact( #TRUE )
      Coil( "Unit1.Em3.ControlNodes".cmCompensatorAxisX.commands.moveVelocity )
   END_RUNG
   // the same network as SCL:
   "Unit1.Em3.ControlNodes".cmCompensatorAxisX.commands.moveVelocity := NOT #TRUE;
END_REGION

REGION Network 53: CmCompensatorAxisX Stop
   RUNG wire#powerrail
      I_Contact( #TRUE )
      Coil( "Unit1.Em3.ControlNodes".cmCompensatorAxisX.commands.stop )
   END_RUNG
   // the same network as SCL:
   "Unit1.Em3.ControlNodes".cmCompensatorAxisX.commands.stop := NOT #TRUE;
END_REGION

REGION Network 54: Call instCmCompensatorAxisX
   RUNG wire#powerrail
      #instCmCompensatorAxisX(enable := TRUE, parentReferenceDesignator := "Unit1.Em3.Config".em.referenceDesignator.combined, enableManualCmds := #statEnableManualCmds, overrideVelocity :=, overrideVelocityPct :=, interlockGeneral := "Unit1.Em3.ControlNodes".cm.Interlock.compensatorAxisX.permit.general, interlockJogForward := "Unit1.Em3.ControlNodes".cm.Interlock.compensatorAxisX.permit.jogForward, interlockJogBackward := "Unit1.Em3.ControlNodes".cm.Interlock.compensatorAxisX.permit.jogBackward, moduleAccessPoint := "BA040AZSCU1~PROFINET_interface~BA040AZSDR3_ModuleAccessPoint", axisNo := 16#6, axis := "Unit1.Em3.Config".axis[1], configuration := "Unit1.Em3.Config".cmCompensatorAxisX, moduleInterface := "Unit1.Em3.HmiInterface".cmCompensatorAxisX, controlNode := "Unit1.Em3.ControlNodes".cmCompensatorAxisX, busy =>, actualPosition =>, actualSpeed =>)
   END_RUNG
   // the same network as SCL:
   #instCmCompensatorAxisX(enable := TRUE,   // "LBC_Axis64Pos_TecPlcCn"
                           parentReferenceDesignator := "Unit1.Em3.Config".em.referenceDesignator.combined,
                           enableManualCmds := #statEnableManualCmds,
                           interlockGeneral := "Unit1.Em3.ControlNodes".cm.Interlock.compensatorAxisX.permit.general,
                           interlockJogForward := "Unit1.Em3.ControlNodes".cm.Interlock.compensatorAxisX.permit.jogForward,
                           interlockJogBackward := "Unit1.Em3.ControlNodes".cm.Interlock.compensatorAxisX.permit.jogBackward,
                           moduleAccessPoint := "BA040AZSCU1~PROFINET_interface~BA040AZSDR3_ModuleAccessPoint",
                           axisNo := 16#6,
                           axis := "Unit1.Em3.Config".axis[1],
                           configuration := "Unit1.Em3.Config".cmCompensatorAxisX,
                           moduleInterface := "Unit1.Em3.HmiInterface".cmCompensatorAxisX,
                           controlNode := "Unit1.Em3.ControlNodes".cmCompensatorAxisX);
END_REGION

REGION Network 55: CmCompensatorAxisX Softcam
   RUNG wire#powerrail
      "LER_SoftCam_Interface_FC"(actualPosition := "Unit1.Em3.HmiInterface".cmCompensatorAxisX.monitoring.actualPosition, selectSetPosition := "Unit1.Em3.HmiInterface".cmCompensatorAxisX.monitoring.selectSetPosition, softCam := "Unit1.Em3.Config".softCam.cmCompensatorAxisX, position := "Unit1.Em3.Config".cmCompensatorAxisX.setPositions, range := 0.01, softCamPos => "Unit1.Em3.ControlNodes".cm.softCam.compensatorAxisX)
   END_RUNG
   // the same network as SCL:
   "LER_SoftCam_Interface_FC"(actualPosition := "Unit1.Em3.HmiInterface".cmCompensatorAxisX.monitoring.actualPosition,
                           selectSetPosition := "Unit1.Em3.HmiInterface".cmCompensatorAxisX.monitoring.selectSetPosition,
                           softCam := "Unit1.Em3.Config".softCam.cmCompensatorAxisX,
                           position := "Unit1.Em3.Config".cmCompensatorAxisX.setPositions,
                           range := 0.01,
                           softCamPos => "Unit1.Em3.ControlNodes".cm.softCam.compensatorAxisX);
END_REGION

REGION Network 56: ********** Control Modules (TwoWayActuator) **********
END_REGION

REGION Network 57: Reset CMS
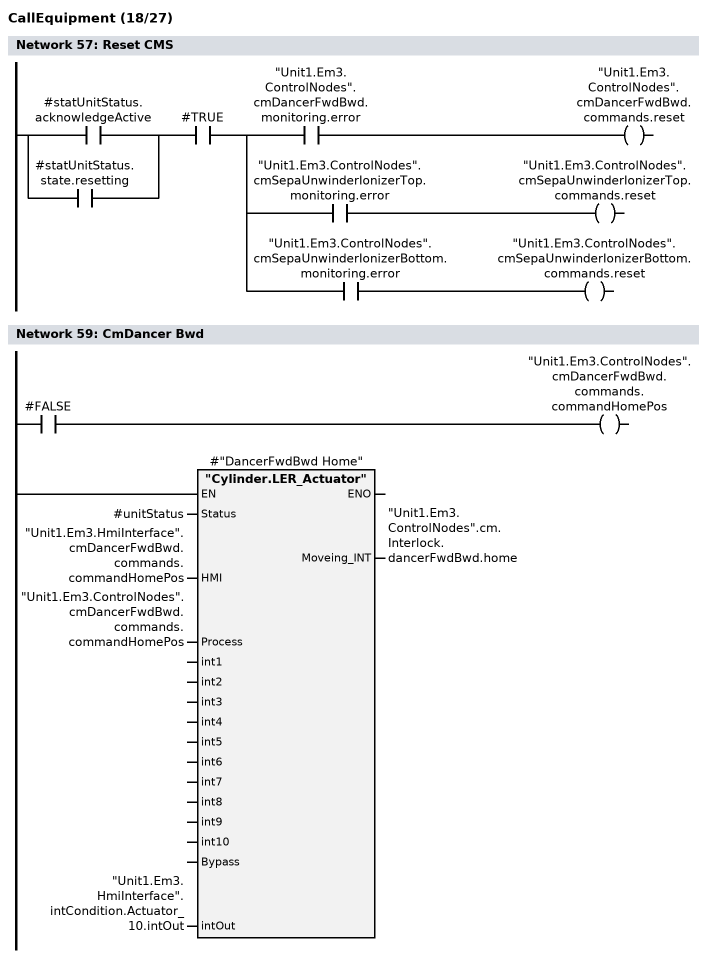
   RUNG wire#powerrail
      Contact( #statUnitStatus.acknowledgeActive )
      wire#w1
      Contact( #TRUE )
      wire#w2
      Contact( "Unit1.Em3.ControlNodes".cmDancerFwdBwd.monitoring.error )
      Coil( "Unit1.Em3.ControlNodes".cmDancerFwdBwd.commands.reset )
   END_RUNG
   RUNG wire#powerrail
      Contact( #statUnitStatus.state.resetting )
   END_RUNG wire#w1
   RUNG wire#w2
      Contact( "Unit1.Em3.ControlNodes".cmSepaUnwinderIonizerTop.monitoring.error )
      Coil( "Unit1.Em3.ControlNodes".cmSepaUnwinderIonizerTop.commands.reset )
   END_RUNG
   RUNG wire#w2
      Contact( "Unit1.Em3.ControlNodes".cmSepaUnwinderIonizerBottom.monitoring.error )
      Coil( "Unit1.Em3.ControlNodes".cmSepaUnwinderIonizerBottom.commands.reset )
   END_RUNG
   // the same network as SCL:
   #_w1 := (#statUnitStatus.acknowledgeActive OR #statUnitStatus.state.resetting) AND #TRUE;
   "Unit1.Em3.ControlNodes".cmDancerFwdBwd.commands.reset := #_w1 AND "Unit1.Em3.ControlNodes".cmDancerFwdBwd.monitoring.error;
   "Unit1.Em3.ControlNodes".cmSepaUnwinderIonizerTop.commands.reset := #_w1 AND "Unit1.Em3.ControlNodes".cmSepaUnwinderIonizerTop.monitoring.error;
   "Unit1.Em3.ControlNodes".cmSepaUnwinderIonizerBottom.commands.reset := #_w1 AND "Unit1.Em3.ControlNodes".cmSepaUnwinderIonizerBottom.monitoring.error;
END_REGION

REGION Network 59: CmDancer Bwd
   RUNG wire#powerrail
      Contact( #FALSE )
      Coil( "Unit1.Em3.ControlNodes".cmDancerFwdBwd.commands.commandHomePos )
   END_RUNG
   RUNG wire#powerrail
      #"DancerFwdBwd Home"(Status := #unitStatus, HMI := "Unit1.Em3.HmiInterface".cmDancerFwdBwd.commands.commandHomePos, Process := "Unit1.Em3.ControlNodes".cmDancerFwdBwd.commands.commandHomePos, int1 :=, int2 :=, int3 :=, int4 :=, int5 :=, int6 :=, int7 :=, int8 :=, int9 :=, int10 :=, Bypass :=, intOut := "Unit1.Em3.HmiInterface".intCondition.Actuator_10.intOut, Moveing_INT => "Unit1.Em3.ControlNodes".cm.Interlock.dancerFwdBwd.home)
   END_RUNG
   // the same network as SCL:
   "Unit1.Em3.ControlNodes".cmDancerFwdBwd.commands.commandHomePos := #FALSE;
   #"DancerFwdBwd Home"(Status := #unitStatus,   // "Cylinder.LER_Actuator"
                        HMI := "Unit1.Em3.HmiInterface".cmDancerFwdBwd.commands.commandHomePos,
                        Process := "Unit1.Em3.ControlNodes".cmDancerFwdBwd.commands.commandHomePos,
                        intOut := "Unit1.Em3.HmiInterface".intCondition.Actuator_10.intOut,
                        Moveing_INT => "Unit1.Em3.ControlNodes".cm.Interlock.dancerFwdBwd.home);
END_REGION

REGION Network 60: CmDancer Fwd
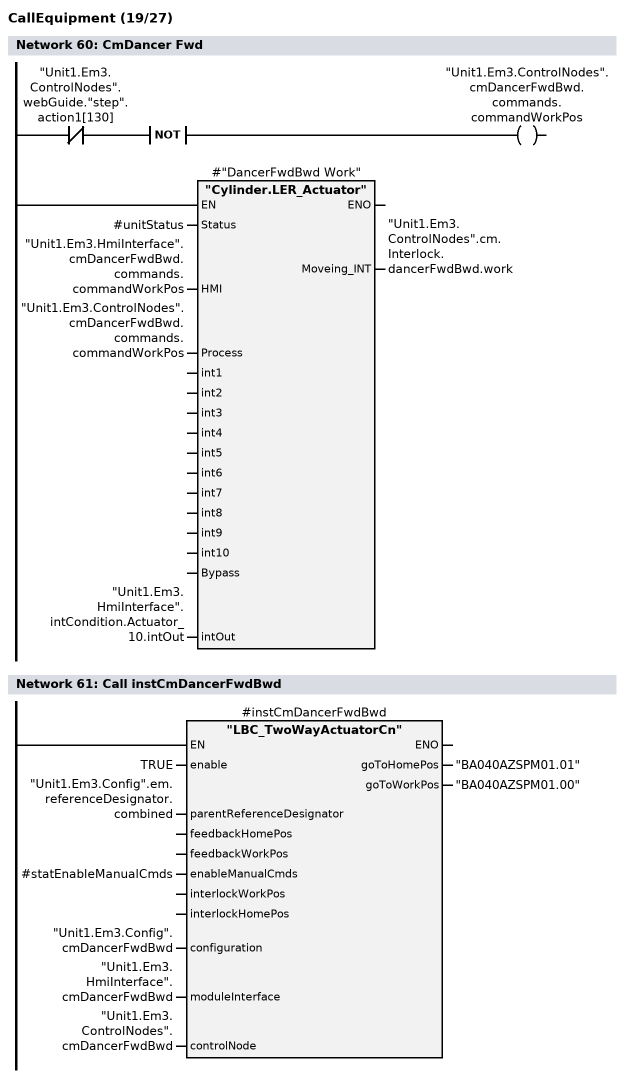
   RUNG wire#powerrail
      I_Contact( "Unit1.Em3.ControlNodes".webGuide."step".action1[130] )
      Not()
      Coil( "Unit1.Em3.ControlNodes".cmDancerFwdBwd.commands.commandWorkPos )
   END_RUNG
   RUNG wire#powerrail
      #"DancerFwdBwd Work"(Status := #unitStatus, HMI := "Unit1.Em3.HmiInterface".cmDancerFwdBwd.commands.commandWorkPos, Process := "Unit1.Em3.ControlNodes".cmDancerFwdBwd.commands.commandWorkPos, int1 :=, int2 :=, int3 :=, int4 :=, int5 :=, int6 :=, int7 :=, int8 :=, int9 :=, int10 :=, Bypass :=, intOut := "Unit1.Em3.HmiInterface".intCondition.Actuator_10.intOut, Moveing_INT => "Unit1.Em3.ControlNodes".cm.Interlock.dancerFwdBwd.work)
   END_RUNG
   // the same network as SCL:
   "Unit1.Em3.ControlNodes".cmDancerFwdBwd.commands.commandWorkPos := NOT (NOT "Unit1.Em3.ControlNodes".webGuide."step".action1[130]);
   #"DancerFwdBwd Work"(Status := #unitStatus,   // "Cylinder.LER_Actuator"
                        HMI := "Unit1.Em3.HmiInterface".cmDancerFwdBwd.commands.commandWorkPos,
                        Process := "Unit1.Em3.ControlNodes".cmDancerFwdBwd.commands.commandWorkPos,
                        intOut := "Unit1.Em3.HmiInterface".intCondition.Actuator_10.intOut,
                        Moveing_INT => "Unit1.Em3.ControlNodes".cm.Interlock.dancerFwdBwd.work);
END_REGION

REGION Network 61: Call instCmDancerFwdBwd
   RUNG wire#powerrail
      #instCmDancerFwdBwd(enable := TRUE, parentReferenceDesignator := "Unit1.Em3.Config".em.referenceDesignator.combined, feedbackHomePos :=, feedbackWorkPos :=, enableManualCmds := #statEnableManualCmds, interlockWorkPos :=, interlockHomePos :=, configuration := "Unit1.Em3.Config".cmDancerFwdBwd, moduleInterface := "Unit1.Em3.HmiInterface".cmDancerFwdBwd, controlNode := "Unit1.Em3.ControlNodes".cmDancerFwdBwd, goToHomePos => "BA040AZSPM01.01", goToWorkPos => "BA040AZSPM01.00")
   END_RUNG
   // the same network as SCL:
   #instCmDancerFwdBwd(enable := TRUE,   // "LBC_TwoWayActuatorCn"
                       parentReferenceDesignator := "Unit1.Em3.Config".em.referenceDesignator.combined,
                       enableManualCmds := #statEnableManualCmds,
                       configuration := "Unit1.Em3.Config".cmDancerFwdBwd,
                       moduleInterface := "Unit1.Em3.HmiInterface".cmDancerFwdBwd,
                       controlNode := "Unit1.Em3.ControlNodes".cmDancerFwdBwd,
                       goToHomePos => "BA040AZSPM01.01",
                       goToWorkPos => "BA040AZSPM01.00");
END_REGION

REGION Network 63: CmSepaUnwinderIonizerTop Home
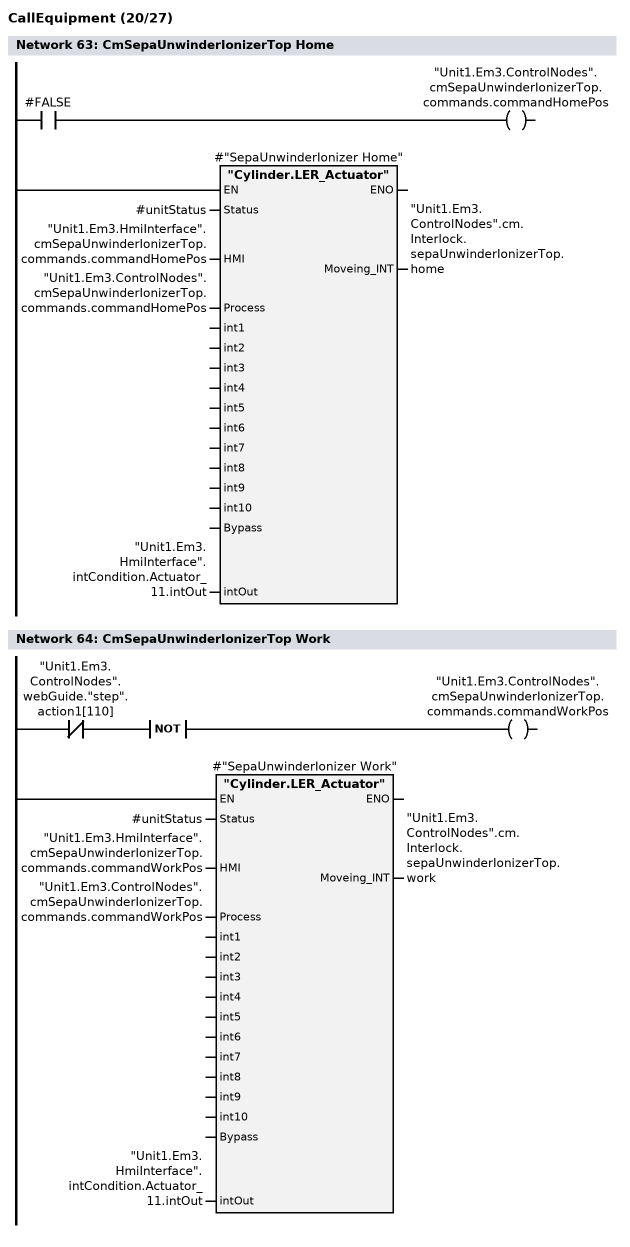
   RUNG wire#powerrail
      Contact( #FALSE )
      Coil( "Unit1.Em3.ControlNodes".cmSepaUnwinderIonizerTop.commands.commandHomePos )
   END_RUNG
   RUNG wire#powerrail
      #"SepaUnwinderIonizer Home"(Status := #unitStatus, HMI := "Unit1.Em3.HmiInterface".cmSepaUnwinderIonizerTop.commands.commandHomePos, Process := "Unit1.Em3.ControlNodes".cmSepaUnwinderIonizerTop.commands.commandHomePos, int1 :=, int2 :=, int3 :=, int4 :=, int5 :=, int6 :=, int7 :=, int8 :=, int9 :=, int10 :=, Bypass :=, intOut := "Unit1.Em3.HmiInterface".intCondition.Actuator_11.intOut, Moveing_INT => "Unit1.Em3.ControlNodes".cm.Interlock.sepaUnwinderIonizerTop.home)
   END_RUNG
   // the same network as SCL:
   "Unit1.Em3.ControlNodes".cmSepaUnwinderIonizerTop.commands.commandHomePos := #FALSE;
   #"SepaUnwinderIonizer Home"(Status := #unitStatus,   // "Cylinder.LER_Actuator"
                           HMI := "Unit1.Em3.HmiInterface".cmSepaUnwinderIonizerTop.commands.commandHomePos,
                           Process := "Unit1.Em3.ControlNodes".cmSepaUnwinderIonizerTop.commands.commandHomePos,
                           intOut := "Unit1.Em3.HmiInterface".intCondition.Actuator_11.intOut,
                           Moveing_INT => "Unit1.Em3.ControlNodes".cm.Interlock.sepaUnwinderIonizerTop.home);
END_REGION

REGION Network 64: CmSepaUnwinderIonizerTop Work
   RUNG wire#powerrail
      I_Contact( "Unit1.Em3.ControlNodes".webGuide."step".action1[110] )
      Not()
      Coil( "Unit1.Em3.ControlNodes".cmSepaUnwinderIonizerTop.commands.commandWorkPos )
   END_RUNG
   RUNG wire#powerrail
      #"SepaUnwinderIonizer Work"(Status := #unitStatus, HMI := "Unit1.Em3.HmiInterface".cmSepaUnwinderIonizerTop.commands.commandWorkPos, Process := "Unit1.Em3.ControlNodes".cmSepaUnwinderIonizerTop.commands.commandWorkPos, int1 :=, int2 :=, int3 :=, int4 :=, int5 :=, int6 :=, int7 :=, int8 :=, int9 :=, int10 :=, Bypass :=, intOut := "Unit1.Em3.HmiInterface".intCondition.Actuator_11.intOut, Moveing_INT => "Unit1.Em3.ControlNodes".cm.Interlock.sepaUnwinderIonizerTop.work)
   END_RUNG
   // the same network as SCL:
   "Unit1.Em3.ControlNodes".cmSepaUnwinderIonizerTop.commands.commandWorkPos := NOT (NOT "Unit1.Em3.ControlNodes".webGuide."step".action1[110]);
   #"SepaUnwinderIonizer Work"(Status := #unitStatus,   // "Cylinder.LER_Actuator"
                           HMI := "Unit1.Em3.HmiInterface".cmSepaUnwinderIonizerTop.commands.commandWorkPos,
                           Process := "Unit1.Em3.ControlNodes".cmSepaUnwinderIonizerTop.commands.commandWorkPos,
                           intOut := "Unit1.Em3.HmiInterface".intCondition.Actuator_11.intOut,
                           Moveing_INT => "Unit1.Em3.ControlNodes".cm.Interlock.sepaUnwinderIonizerTop.work);
END_REGION

REGION Network 65: Call instCmSepaUnwinderIonizerTop
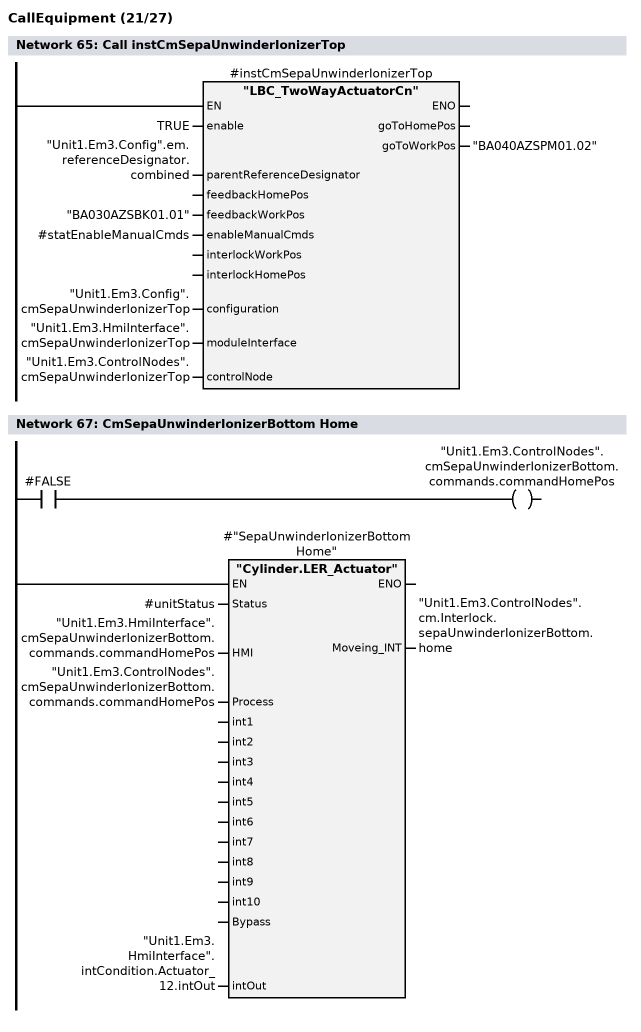
   RUNG wire#powerrail
      #instCmSepaUnwinderIonizerTop(enable := TRUE, parentReferenceDesignator := "Unit1.Em3.Config".em.referenceDesignator.combined, feedbackHomePos :=, feedbackWorkPos := "BA030AZSBK01.01", enableManualCmds := #statEnableManualCmds, interlockWorkPos :=, interlockHomePos :=, configuration := "Unit1.Em3.Config".cmSepaUnwinderIonizerTop, moduleInterface := "Unit1.Em3.HmiInterface".cmSepaUnwinderIonizerTop, controlNode := "Unit1.Em3.ControlNodes".cmSepaUnwinderIonizerTop, goToHomePos =>, goToWorkPos => "BA040AZSPM01.02")
   END_RUNG
   // the same network as SCL:
   #instCmSepaUnwinderIonizerTop(enable := TRUE,   // "LBC_TwoWayActuatorCn"
                           parentReferenceDesignator := "Unit1.Em3.Config".em.referenceDesignator.combined,
                           feedbackWorkPos := "BA030AZSBK01.01",
                           enableManualCmds := #statEnableManualCmds,
                           configuration := "Unit1.Em3.Config".cmSepaUnwinderIonizerTop,
                           moduleInterface := "Unit1.Em3.HmiInterface".cmSepaUnwinderIonizerTop,
                           controlNode := "Unit1.Em3.ControlNodes".cmSepaUnwinderIonizerTop,
                           goToWorkPos => "BA040AZSPM01.02");
END_REGION

REGION Network 67: CmSepaUnwinderIonizerBottom Home
   RUNG wire#powerrail
      Contact( #FALSE )
      Coil( "Unit1.Em3.ControlNodes".cmSepaUnwinderIonizerBottom.commands.commandHomePos )
   END_RUNG
   RUNG wire#powerrail
      #"SepaUnwinderIonizerBottom Home"(Status := #unitStatus, HMI := "Unit1.Em3.HmiInterface".cmSepaUnwinderIonizerBottom.commands.commandHomePos, Process := "Unit1.Em3.ControlNodes".cmSepaUnwinderIonizerBottom.commands.commandHomePos, int1 :=, int2 :=, int3 :=, int4 :=, int5 :=, int6 :=, int7 :=, int8 :=, int9 :=, int10 :=, Bypass :=, intOut := "Unit1.Em3.HmiInterface".intCondition.Actuator_12.intOut, Moveing_INT => "Unit1.Em3.ControlNodes".cm.Interlock.sepaUnwinderIonizerBottom.home)
   END_RUNG
   // the same network as SCL:
   "Unit1.Em3.ControlNodes".cmSepaUnwinderIonizerBottom.commands.commandHomePos := #FALSE;
   #"SepaUnwinderIonizerBottom Home"(Status := #unitStatus,   // "Cylinder.LER_Actuator"
                           HMI := "Unit1.Em3.HmiInterface".cmSepaUnwinderIonizerBottom.commands.commandHomePos,
                           Process := "Unit1.Em3.ControlNodes".cmSepaUnwinderIonizerBottom.commands.commandHomePos,
                           intOut := "Unit1.Em3.HmiInterface".intCondition.Actuator_12.intOut,
                           Moveing_INT => "Unit1.Em3.ControlNodes".cm.Interlock.sepaUnwinderIonizerBottom.home);
END_REGION

REGION Network 68: CmSepaUnwinderIonizerBottom Work
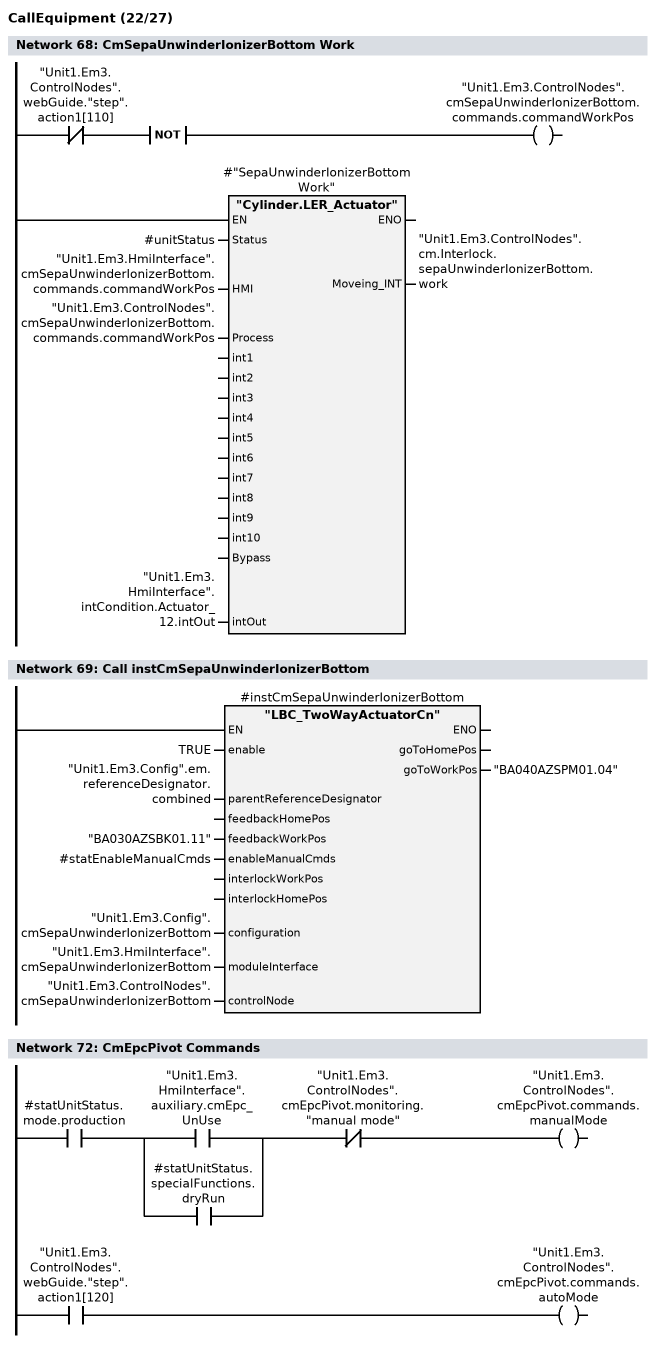
   RUNG wire#powerrail
      I_Contact( "Unit1.Em3.ControlNodes".webGuide."step".action1[110] )
      Not()
      Coil( "Unit1.Em3.ControlNodes".cmSepaUnwinderIonizerBottom.commands.commandWorkPos )
   END_RUNG
   RUNG wire#powerrail
      #"SepaUnwinderIonizerBottom Work"(Status := #unitStatus, HMI := "Unit1.Em3.HmiInterface".cmSepaUnwinderIonizerBottom.commands.commandWorkPos, Process := "Unit1.Em3.ControlNodes".cmSepaUnwinderIonizerBottom.commands.commandWorkPos, int1 :=, int2 :=, int3 :=, int4 :=, int5 :=, int6 :=, int7 :=, int8 :=, int9 :=, int10 :=, Bypass :=, intOut := "Unit1.Em3.HmiInterface".intCondition.Actuator_12.intOut, Moveing_INT => "Unit1.Em3.ControlNodes".cm.Interlock.sepaUnwinderIonizerBottom.work)
   END_RUNG
   // the same network as SCL:
   "Unit1.Em3.ControlNodes".cmSepaUnwinderIonizerBottom.commands.commandWorkPos := NOT (NOT "Unit1.Em3.ControlNodes".webGuide."step".action1[110]);
   #"SepaUnwinderIonizerBottom Work"(Status := #unitStatus,   // "Cylinder.LER_Actuator"
                           HMI := "Unit1.Em3.HmiInterface".cmSepaUnwinderIonizerBottom.commands.commandWorkPos,
                           Process := "Unit1.Em3.ControlNodes".cmSepaUnwinderIonizerBottom.commands.commandWorkPos,
                           intOut := "Unit1.Em3.HmiInterface".intCondition.Actuator_12.intOut,
                           Moveing_INT => "Unit1.Em3.ControlNodes".cm.Interlock.sepaUnwinderIonizerBottom.work);
END_REGION

REGION Network 69: Call instCmSepaUnwinderIonizerBottom
   RUNG wire#powerrail
      #instCmSepaUnwinderIonizerBottom(enable := TRUE, parentReferenceDesignator := "Unit1.Em3.Config".em.referenceDesignator.combined, feedbackHomePos :=, feedbackWorkPos := "BA030AZSBK01.11", enableManualCmds := #statEnableManualCmds, interlockWorkPos :=, interlockHomePos :=, configuration := "Unit1.Em3.Config".cmSepaUnwinderIonizerBottom, moduleInterface := "Unit1.Em3.HmiInterface".cmSepaUnwinderIonizerBottom, controlNode := "Unit1.Em3.ControlNodes".cmSepaUnwinderIonizerBottom, goToHomePos =>, goToWorkPos => "BA040AZSPM01.04")
   END_RUNG
   // the same network as SCL:
   #instCmSepaUnwinderIonizerBottom(enable := TRUE,   // "LBC_TwoWayActuatorCn"
                           parentReferenceDesignator := "Unit1.Em3.Config".em.referenceDesignator.combined,
                           feedbackWorkPos := "BA030AZSBK01.11",
                           enableManualCmds := #statEnableManualCmds,
                           configuration := "Unit1.Em3.Config".cmSepaUnwinderIonizerBottom,
                           moduleInterface := "Unit1.Em3.HmiInterface".cmSepaUnwinderIonizerBottom,
                           controlNode := "Unit1.Em3.ControlNodes".cmSepaUnwinderIonizerBottom,
                           goToWorkPos => "BA040AZSPM01.04");
END_REGION

REGION Network 70: ******************** Control Modules (Accessories) ********************
END_REGION

REGION Network 71: Reset CMS
END_REGION

REGION Network 72: CmEpcPivot Commands
   RUNG wire#powerrail
      Contact( #statUnitStatus.mode.production )
      wire#w1
      Contact( "Unit1.Em3.HmiInterface".auxiliary.cmEpc_UnUse )
      wire#w2
      I_Contact( "Unit1.Em3.ControlNodes".cmEpcPivot.monitoring."manual mode" )
      Coil( "Unit1.Em3.ControlNodes".cmEpcPivot.commands.manualMode )
   END_RUNG
   RUNG wire#w1
      Contact( #statUnitStatus.specialFunctions.dryRun )
   END_RUNG wire#w2
   RUNG wire#powerrail
      Contact( "Unit1.Em3.ControlNodes".webGuide."step".action1[120] )
      Coil( "Unit1.Em3.ControlNodes".cmEpcPivot.commands.autoMode )
   END_RUNG
   // the same network as SCL:
   "Unit1.Em3.ControlNodes".cmEpcPivot.commands.manualMode := #statUnitStatus.mode.production AND ("Unit1.Em3.HmiInterface".auxiliary.cmEpc_UnUse OR #statUnitStatus.specialFunctions.dryRun) AND NOT "Unit1.Em3.ControlNodes".cmEpcPivot.monitoring."manual mode";
   "Unit1.Em3.ControlNodes".cmEpcPivot.commands.autoMode := "Unit1.Em3.ControlNodes".webGuide."step".action1[120];
END_REGION

REGION Network 73: Call instCmEpcPivot
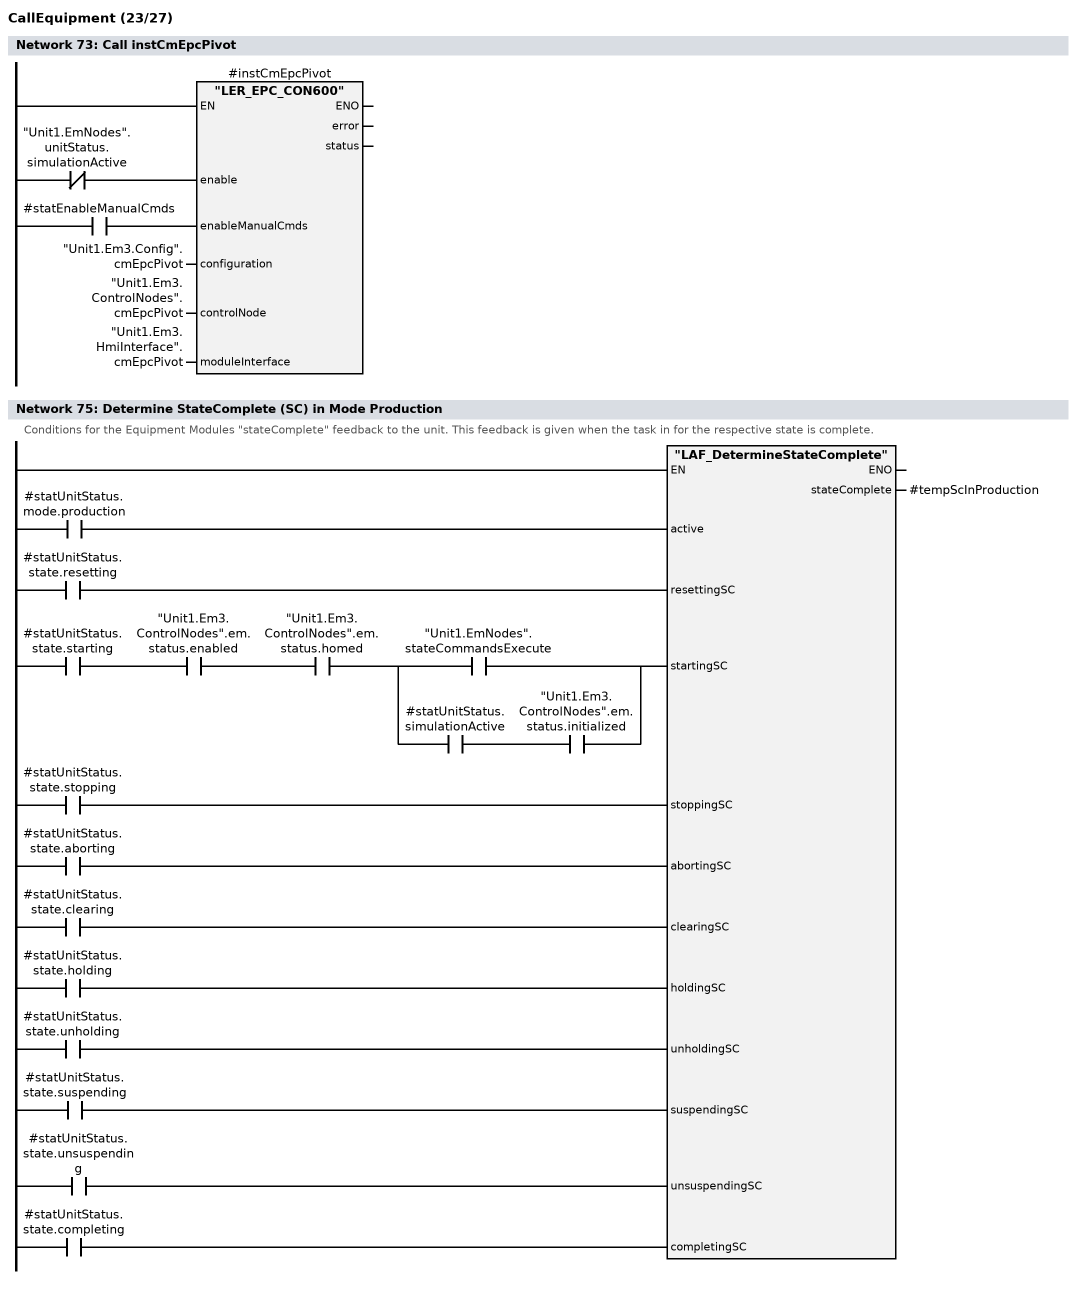
   RUNG wire#powerrail
      #instCmEpcPivot(enable := wire#w1, enableManualCmds := wire#w2, configuration := "Unit1.Em3.Config".cmEpcPivot, controlNode := "Unit1.Em3.ControlNodes".cmEpcPivot, moduleInterface := "Unit1.Em3.HmiInterface".cmEpcPivot, error =>, status =>)
   END_RUNG
   RUNG wire#powerrail
      I_Contact( "Unit1.EmNodes".unitStatus.simulationActive )
   END_RUNG wire#w1
   RUNG wire#powerrail
      Contact( #statEnableManualCmds )
   END_RUNG wire#w2
   // the same network as SCL:
   #instCmEpcPivot(enable := NOT "Unit1.EmNodes".unitStatus.simulationActive,   // "LER_EPC_CON600"
                   enableManualCmds := #statEnableManualCmds,
                   configuration := "Unit1.Em3.Config".cmEpcPivot,
                   controlNode := "Unit1.Em3.ControlNodes".cmEpcPivot,
                   moduleInterface := "Unit1.Em3.HmiInterface".cmEpcPivot);
END_REGION

REGION Network 74: *************** Feedback to Unit ***************************
END_REGION

REGION Network 75: Determine StateComplete (SC) in Mode Production
   // Conditions for the Equipment Modules "stateComplete" feedback to the unit. This feedback is given when the task in for the respective state is complete.
   RUNG wire#powerrail
      "LAF_DetermineStateComplete"(active := wire#w1, resettingSC := wire#w2, startingSC := wire#w4, stoppingSC := wire#w5, abortingSC := wire#w6, clearingSC := wire#w7, holdingSC := wire#w8, unholdingSC := wire#w9, suspendingSC := wire#w10, unsuspendingSC := wire#w11, completingSC := wire#w12, stateComplete => #tempScInProduction)
   END_RUNG
   RUNG wire#powerrail
      Contact( #statUnitStatus.mode.production )
   END_RUNG wire#w1
   RUNG wire#powerrail
      Contact( #statUnitStatus.state.resetting )
   END_RUNG wire#w2
   RUNG wire#powerrail
      Contact( #statUnitStatus.state.starting )
      Contact( "Unit1.Em3.ControlNodes".em.status.enabled )
      Contact( "Unit1.Em3.ControlNodes".em.status.homed )
      wire#w3
      Contact( "Unit1.EmNodes".stateCommandsExecute )
   END_RUNG wire#w4
   RUNG wire#w3
      Contact( #statUnitStatus.simulationActive )
      Contact( "Unit1.Em3.ControlNodes".em.status.initialized )
   END_RUNG wire#w4
   RUNG wire#powerrail
      Contact( #statUnitStatus.state.stopping )
   END_RUNG wire#w5
   RUNG wire#powerrail
      Contact( #statUnitStatus.state.aborting )
   END_RUNG wire#w6
   RUNG wire#powerrail
      Contact( #statUnitStatus.state.clearing )
   END_RUNG wire#w7
   RUNG wire#powerrail
      Contact( #statUnitStatus.state.holding )
   END_RUNG wire#w8
   RUNG wire#powerrail
      Contact( #statUnitStatus.state.unholding )
   END_RUNG wire#w9
   RUNG wire#powerrail
      Contact( #statUnitStatus.state.suspending )
   END_RUNG wire#w10
   RUNG wire#powerrail
      Contact( #statUnitStatus.state.unsuspending )
   END_RUNG wire#w11
   RUNG wire#powerrail
      Contact( #statUnitStatus.state.completing )
   END_RUNG wire#w12
   // the same network as SCL:
   "LAF_DetermineStateComplete"(active := #statUnitStatus.mode.production,
                           resettingSC := #statUnitStatus.state.resetting,
                           startingSC := #statUnitStatus.state.starting AND "Unit1.Em3.ControlNodes".em.status.enabled AND "Unit1.Em3.ControlNodes".em.status.homed AND ("Unit1.EmNodes".stateCommandsExecute OR (#statUnitStatus.simulationActive AND "Unit1.Em3.ControlNodes".em.status.initialized)),
                           stoppingSC := #statUnitStatus.state.stopping,
                           abortingSC := #statUnitStatus.state.aborting,
                           clearingSC := #statUnitStatus.state.clearing,
                           holdingSC := #statUnitStatus.state.holding,
                           unholdingSC := #statUnitStatus.state.unholding,
                           suspendingSC := #statUnitStatus.state.suspending,
                           unsuspendingSC := #statUnitStatus.state.unsuspending,
                           completingSC := #statUnitStatus.state.completing,
                           stateComplete => #tempScInProduction);
END_REGION

REGION Network 76: Determine StateComplete (SC) in Mode Maintenance/Manual
   // Conditions for the Equipment Modules "stateComplete" feedback to the unit. This feedback is given when the task in for the respective state is complete.
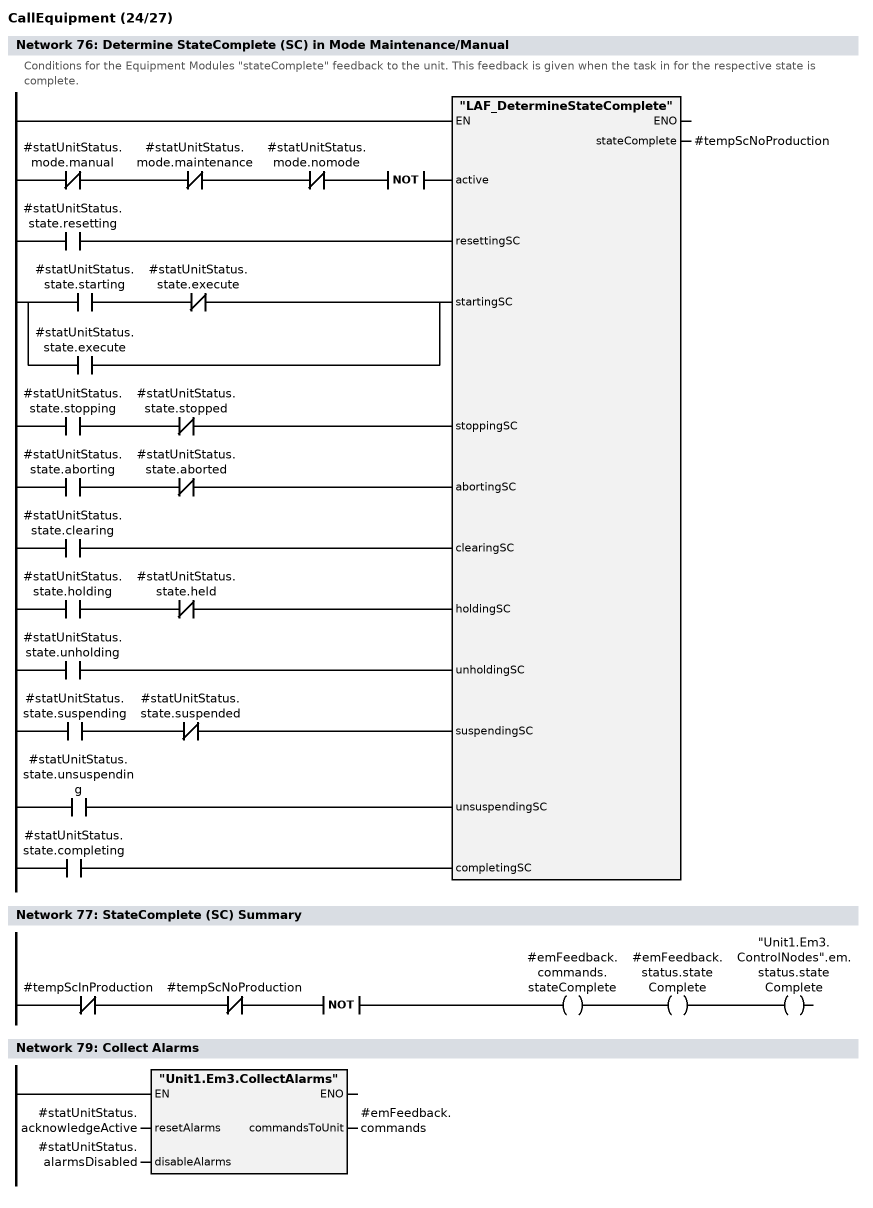
   RUNG wire#powerrail
      "LAF_DetermineStateComplete"(active := wire#w1, resettingSC := wire#w2, startingSC := wire#w3, stoppingSC := wire#w4, abortingSC := wire#w5, clearingSC := wire#w6, holdingSC := wire#w7, unholdingSC := wire#w8, suspendingSC := wire#w9, unsuspendingSC := wire#w10, completingSC := wire#w11, stateComplete => #tempScNoProduction)
   END_RUNG
   RUNG wire#powerrail
      I_Contact( #statUnitStatus.mode.manual )
      I_Contact( #statUnitStatus.mode.maintenance )
      I_Contact( #statUnitStatus.mode.nomode )
      Not()
   END_RUNG wire#w1
   RUNG wire#powerrail
      Contact( #statUnitStatus.state.resetting )
   END_RUNG wire#w2
   RUNG wire#powerrail
      Contact( #statUnitStatus.state.starting )
      I_Contact( #statUnitStatus.state.execute )
   END_RUNG wire#w3
   RUNG wire#powerrail
      Contact( #statUnitStatus.state.execute )
   END_RUNG wire#w3
   RUNG wire#powerrail
      Contact( #statUnitStatus.state.stopping )
      I_Contact( #statUnitStatus.state.stopped )
   END_RUNG wire#w4
   RUNG wire#powerrail
      Contact( #statUnitStatus.state.aborting )
      I_Contact( #statUnitStatus.state.aborted )
   END_RUNG wire#w5
   RUNG wire#powerrail
      Contact( #statUnitStatus.state.clearing )
   END_RUNG wire#w6
   RUNG wire#powerrail
      Contact( #statUnitStatus.state.holding )
      I_Contact( #statUnitStatus.state.held )
   END_RUNG wire#w7
   RUNG wire#powerrail
      Contact( #statUnitStatus.state.unholding )
   END_RUNG wire#w8
   RUNG wire#powerrail
      Contact( #statUnitStatus.state.suspending )
      I_Contact( #statUnitStatus.state.suspended )
   END_RUNG wire#w9
   RUNG wire#powerrail
      Contact( #statUnitStatus.state.unsuspending )
   END_RUNG wire#w10
   RUNG wire#powerrail
      Contact( #statUnitStatus.state.completing )
   END_RUNG wire#w11
   // the same network as SCL:
   "LAF_DetermineStateComplete"(active := NOT (NOT #statUnitStatus.mode.manual AND NOT #statUnitStatus.mode.maintenance AND NOT #statUnitStatus.mode.nomode),
                           resettingSC := #statUnitStatus.state.resetting,
                           startingSC := (#statUnitStatus.state.starting AND NOT #statUnitStatus.state.execute) OR #statUnitStatus.state.execute,
                           stoppingSC := #statUnitStatus.state.stopping AND NOT #statUnitStatus.state.stopped,
                           abortingSC := #statUnitStatus.state.aborting AND NOT #statUnitStatus.state.aborted,
                           clearingSC := #statUnitStatus.state.clearing,
                           holdingSC := #statUnitStatus.state.holding AND NOT #statUnitStatus.state.held,
                           unholdingSC := #statUnitStatus.state.unholding,
                           suspendingSC := #statUnitStatus.state.suspending AND NOT #statUnitStatus.state.suspended,
                           unsuspendingSC := #statUnitStatus.state.unsuspending,
                           completingSC := #statUnitStatus.state.completing,
                           stateComplete => #tempScNoProduction);
END_REGION

REGION Network 77: StateComplete (SC) Summary
   RUNG wire#powerrail
      I_Contact( #tempScInProduction )
      I_Contact( #tempScNoProduction )
      Not()
      Coil( #emFeedback.commands.stateComplete )
      Coil( #emFeedback.status.stateComplete )
      Coil( "Unit1.Em3.ControlNodes".em.status.stateComplete )
   END_RUNG
   // the same network as SCL:
   #emFeedback.commands.stateComplete := NOT (NOT #tempScInProduction AND NOT #tempScNoProduction);
   #emFeedback.status.stateComplete := #emFeedback.commands.stateComplete;
   "Unit1.Em3.ControlNodes".em.status.stateComplete := #emFeedback.commands.stateComplete;
END_REGION

REGION Network 78: *************** Alarms **********************************
END_REGION

REGION Network 79: Collect Alarms
   RUNG wire#powerrail
      "Unit1.Em3.CollectAlarms"(resetAlarms := #statUnitStatus.acknowledgeActive, disableAlarms := #statUnitStatus.alarmsDisabled, commandsToUnit => #emFeedback.commands)
   END_RUNG
   // the same network as SCL:
   "Unit1.Em3.CollectAlarms"(resetAlarms := #statUnitStatus.acknowledgeActive,
                           disableAlarms := #statUnitStatus.alarmsDisabled,
                           commandsToUnit => #emFeedback.commands);
END_REGION

REGION Network 80: Manage Alarms
   // Derive commands from the ProDiag supervision. The ProDiag supervisions contain categories which define the reaction of these supervisions (e.g. abort, stop, hold). These are handed over as commands to the unit level.
   // Alternatively, if no ProDiag should be used, you can use the LAF_ManageBitAlarms to realize bit alarm handling. This block can be found in LAF in folder 70_AlarmHandling.
